(* IEC 61131-3 sources: PortalRobot/Portal_robot/Device/application/FB, 34 files *)

(* ---- FB_ALARM_MANAGER.st ---- *)
FUNCTION_BLOCK FB_ALARM_MANAGER
VAR_INPUT
	xResetAll      : BOOL; // Общий сброс ошибок ячейки
	xResetWarnings : BOOL; // Сброс накопленных предупреждений
END_VAR
VAR_IN_OUT
	Sources : ARRAY [1..13] OF ST_ALARM_SOURCE_DATA; // Унифицированные данные функциональных блоков
END_VAR
VAR_OUTPUT
	Status : ST_ALARM_STATUS; // Сводный статус журнала
	Events : ARRAY [1..100] OF ST_ALARM_EVENT; // Журнал активных и зафиксированных событий
END_VAR
VAR
	uiWriteIndex : UINT := 1; // Следующая ячейка кольцевого журнала
	udiSequence  : UDINT; // Общий порядковый номер события
	adwPreviousAlarm : ARRAY [1..13] OF DWORD; // Опубликованные аварии прошлого цикла
	audiPreviousWarning : ARRAY [1..13] OF UDINT; // Номера предупреждений прошлого цикла
	uiIndex : UINT; // Индекс источника или события
END_VAR

// --- BEGIN IMPLEMENTATION ---

// Предупреждения подтверждаются отдельно или вместе с общим сбросом.
IF xResetWarnings OR xResetAll THEN
	FOR uiIndex := 1 TO 100 DO
		IF Events[uiIndex].xActive
		AND (Events[uiIndex].eSeverity = E_ALARM_SEVERITY.WARNING) THEN
			Events[uiIndex].xActive := FALSE;
		END_IF;
	END_FOR;
END_IF;

// Менеджер не определяет причины: он регистрирует подготовленные данные владельцев блоков.
FOR uiIndex := 1 TO 13 DO
	UpdateSource(
		eSource := Sources[uiIndex].eSource,
		dwCurrent := Sources[uiIndex].dwAlarmActive,
		dwPrevious := adwPreviousAlarm[uiIndex]
	);

	IF Sources[uiIndex].stWarning.udiSequence <> audiPreviousWarning[uiIndex] THEN
		IF (Sources[uiIndex].stWarning.udiSequence <> UDINT#0)
		AND (Sources[uiIndex].stWarning.uiCode <> UINT#0) THEN
			AddEvent(
				eSource := Sources[uiIndex].eSource,
				eSeverity := E_ALARM_SEVERITY.WARNING,
				uiCode := Sources[uiIndex].stWarning.uiCode
			);
		END_IF;
		audiPreviousWarning[uiIndex] := Sources[uiIndex].stWarning.udiSequence;
	END_IF;
END_FOR;

Status.uiActiveAlarmCount := 0;
Status.uiActiveWarningCount := 0;
Status.uiHistoryCount := 0;

FOR uiIndex := 1 TO 100 DO
	IF Events[uiIndex].udiSequence <> UDINT#0 THEN
		Status.uiHistoryCount := Status.uiHistoryCount + 1;
	END_IF;
	IF Events[uiIndex].xActive THEN
		IF Events[uiIndex].eSeverity = E_ALARM_SEVERITY.ALARM THEN
			Status.uiActiveAlarmCount := Status.uiActiveAlarmCount + 1;
		ELSE
			Status.uiActiveWarningCount := Status.uiActiveWarningCount + 1;
		END_IF;
	END_IF;
END_FOR;

Status.uiActiveEventCount := Status.uiActiveAlarmCount + Status.uiActiveWarningCount;
Status.xAlarmActive := Status.uiActiveAlarmCount > 0;
Status.xWarningActive := Status.uiActiveWarningCount > 0;

(* ---- FB_AXIS.st ---- *)
FUNCTION_BLOCK FB_Axis
VAR_IN_OUT
    Axis     : AXIS_REF_SM3;   // ссылка на ось SoftMotion
    AxisData : ST_AXIS;        // все данные оси (команды, параметры, статусы)
END_VAR

VAR CONSTANT
    // ==================================================
    // Ошибки оси, MC-блоков и SoftMotion
    // ==================================================
    AXE_MC_POWER_ERROR       : DWORD := DWORD#16#00000001; // Ошибка MC_Power
    AXE_MC_RESET_ERROR       : DWORD := DWORD#16#00000002; // Ошибка MC_Reset
    AXE_MC_STOP_ERROR        : DWORD := DWORD#16#00000004; // Ошибка MC_Stop
    AXE_MC_JOG_ERROR         : DWORD := DWORD#16#00000008; // Ошибка MC_Jog
    AXE_MC_HOME_ERROR        : DWORD := DWORD#16#00000010; // Ошибка MC_Home
    AXE_MC_MOVE_ABS_ERROR    : DWORD := DWORD#16#00000020; // Ошибка абсолютного перемещения
    AXE_MC_MOVE_REL_ERROR    : DWORD := DWORD#16#00000040; // Ошибка относительного перемещения
    AXE_READ_POS_ERROR       : DWORD := DWORD#16#00000080; // Ошибка чтения позиции
    AXE_READ_STATUS_ERROR    : DWORD := DWORD#16#00000100; // Ошибка чтения статуса
    AXE_ERRORSTOP            : DWORD := DWORD#16#00000200; // Ось находится в ErrorStop
    AXE_FB_ERROR_OCCURRED    : DWORD := DWORD#16#00000400; // SoftMotion сообщил внутреннюю ошибку
    AXE_COMMAND_ABORTED      : DWORD := DWORD#16#00000800; // Команда движения прервана
    AXE_UNKNOWN_ACTUAL_ERROR : DWORD := DWORD#16#00001000; // Неизвестная текущая ошибка
    AXE_DRIVE_AXIS_ERROR     : DWORD := DWORD#16#00002000; // Ошибка привода

    // ==================================================
    // Логические ошибки блока
    // ==================================================
    LOG_POWER_PERMIT_LOST    : DWORD := DWORD#16#00000001; // Снято разрешение питания
    LOG_GLOBAL_DURING_POWER  : DWORD := DWORD#16#00000002; // Глобальная ошибка при включении
    LOG_GLOBAL_DURING_READY  : DWORD := DWORD#16#00000004; // Глобальная ошибка в готовности
    LOG_GLOBAL_DURING_MOTION : DWORD := DWORD#16#00000008; // Глобальная ошибка при движении
    LOG_JOG_CONFLICT         : DWORD := DWORD#16#00000010; // Одновременно заданы Jog+ и Jog-
    LOG_MOVE_ABS_NOT_HOMED   : DWORD := DWORD#16#00000020; // Абсолютное движение без поиска дома
    LOG_MOVE_REL_NOT_HOMED   : DWORD := DWORD#16#00000040; // Относительное движение без поиска дома
    LOG_STEP_TIMEOUT         : DWORD := DWORD#16#00000080; // Превышено время шага
    LOG_UNKNOWN_STEP         : DWORD := DWORD#16#00000100; // Неизвестный шаг автомата

    // ==================================================
    // Предупреждения блока
    // ==================================================
    WRN_NO_POWER_PERMIT : DWORD := DWORD#16#00000001; // Нет разрешения подачи питания

    MASK_LOCAL_LOGICAL_ERROR : DWORD :=
        LOG_JOG_CONFLICT OR
        LOG_MOVE_ABS_NOT_HOMED OR
        LOG_MOVE_REL_NOT_HOMED OR
        LOG_STEP_TIMEOUT OR
        LOG_UNKNOWN_STEP; // Логические первопричины, принадлежащие оси
END_VAR

VAR
    // Триггеры на команды
    rtEnable            : R_TRIG; // Фронт команды включения
    rtDisable           : R_TRIG; // Фронт команды отключения
    rtResetAllError     : R_TRIG; // Фронт общего сброса
    rtResetAxisError    : R_TRIG; // Фронт сброса привода
    rtResetLogicalError : R_TRIG; // Фронт сброса логики
    rtStop              : R_TRIG; // Фронт команды остановки
    rtHome              : R_TRIG; // Фронт команды поиска дома
    rtMoveAbsolute      : R_TRIG; // Фронт абсолютного перемещения
    rtMoveRelative      : R_TRIG; // Фронт относительного перемещения

    // Экземпляры MC-блоков
    fbPower        : MC_Power; // Управление питанием привода
    fbReset        : MC_Reset; // Сброс ошибки привода
    fbStop         : MC_Stop; // Контролируемая остановка
    fbJog          : MC_Jog; // Толчковое движение
    fbHome         : MC_Home; // Поиск домашней позиции
    fbMoveAbsolute : MC_MoveAbsolute; // Абсолютное перемещение
    fbMoveRelative : MC_MoveRelative; // Относительное перемещение
    fbReadPosition : MC_ReadActualPosition; // Чтение текущей позиции
    fbReadStatus   : MC_ReadStatus; // Чтение состояния оси
    fbReadAxisError: MC_ReadAxisError; // Чтение кода ошибки привода

    // Внутренние управляющие флаги
    xPowerRequest    : BOOL; // Защёлкнутый запрос питания
    xResetExecute    : BOOL; // Выполняется сброс привода
    xStopExecute     : BOOL; // Выполняется остановка
    xHomeExecute     : BOOL; // Выполняется поиск дома
    xMoveAbsExecute  : BOOL; // Выполняется абсолютное перемещение
    xMoveRelExecute  : BOOL; // Выполняется относительное перемещение
    xJogForwardExec  : BOOL; // Выполняется Jog в положительную сторону
    xJogBackwardExec : BOOL; // Выполняется Jog в отрицательную сторону

    // Для таймера шага
    iPrevStep        : E_AXIS_STATE := E_AXIS_STATE.DISABLED; // Предыдущий шаг автомата
    xStepChanged     : BOOL; // Шаг изменился в текущем цикле
    xStepTimerEnable : BOOL; // Разрешение таймера шага
    tonStep          : TON; // Таймер времени на шаге
    tonStepTimeout   : TON; // Таймер превышения времени шага

    // Для удержания предупреждений
    tpWarningHold : TP; // Удержание предупреждения для отображения
    xWarningPulse : BOOL; // Импульс нового предупреждения

    // Вспомогательные флаги для сброса
    xDoResetAxis    : BOOL; // Требуется сброс ошибок привода
    xDoResetLogical : BOOL; // Требуется сброс логических ошибок
    xNeedMcReset    : BOOL; // Требуется вызов MC_Reset

    // Актуальная ошибка оси (на основе MC-блоков)
    xAxisErrorActual : BOOL; // Текущая ошибка по выходам MC-блоков
END_VAR

// --- BEGIN IMPLEMENTATION ---

// ======================================================
// 1. ФРОНТЫ (триггеры на команды из структуры)
// ======================================================
rtEnable(CLK := AxisData.Command.xEnable);
rtDisable(CLK := AxisData.Command.xDisable);
rtResetAllError(CLK := AxisData.Command.xResetAllError);
rtResetAxisError(CLK := AxisData.Command.xResetAxisError);
rtResetLogicalError(CLK := AxisData.Command.xResetLogicalError);
rtStop(CLK := AxisData.Command.xStop);
rtHome(CLK := AxisData.Command.xHome);
rtMoveAbsolute(CLK := AxisData.Command.xMoveAbsolute);
rtMoveRelative(CLK := AxisData.Command.xMoveRelative);

// ======================================================
// 2. СТАТУСЫ ОТ MC-БЛОКОВ (запись в структуру)
// ======================================================
AxisData.Status.xPowered := fbPower.Status;

AxisData.Status.xLocalError :=
    fbPower.Error OR
    fbReset.Error OR
    fbStop.Error OR
    fbJog.Error OR
    fbHome.Error OR
    fbMoveAbsolute.Error OR
    fbMoveRelative.Error OR
    fbReadPosition.Error OR
    fbReadStatus.Error OR
    fbReadStatus.Errorstop OR
    fbReadStatus.FBErrorOccured;

AxisData.Status.xMotionBusy :=
    fbStop.Busy OR
    fbJog.Busy OR
    fbHome.Busy OR
    fbMoveAbsolute.Busy OR
    fbMoveRelative.Busy;

// MC_Reset нужен только для аппаратных/SoftMotion ошибок
xNeedMcReset := fbReadStatus.Errorstop OR fbReadStatus.FBErrorOccured OR fbReadAxisError.AxisError;

AxisData.Error.dwAxisError := AxisData.Error.dwAxisErrorActual OR AxisData.Error.dwAxisErrorLatched;
AxisData.Error.dwLogicalError := AxisData.Error.dwLogicalErrorLatched;
AxisData.Error.dwAllError := AxisData.Error.dwAxisError OR AxisData.Error.dwLogicalError;

// ======================================================
// 3. ЗНАЧЕНИЯ ПО УМОЛЧАНИЮ ДЛЯ ИСПОЛНИТЕЛЬНЫХ ФЛАГОВ
// ======================================================
xResetExecute    := FALSE;
xStopExecute     := FALSE;
xHomeExecute     := FALSE;
xMoveAbsExecute  := FALSE;
xMoveRelExecute  := FALSE;
xJogForwardExec  := FALSE;
xJogBackwardExec := FALSE;

AxisData.Status.xDone := FALSE;
xWarningPulse := FALSE;

// ======================================================
// 4. КОНЕЧНЫЙ АВТОМАТ (используем перечисление E_AXIS_STATE)
// ======================================================
CASE AxisData.Diag.iStep OF

    // --------------------------------------------------
    E_AXIS_STATE.DISABLED:
    // --------------------------------------------------
        AxisData.Diag.sStepName := 'DISABLED';
        AxisData.Diag.sWaitReason := 'Waiting Enable command';
        AxisData.Diag.tStepPreset := T#0S;

        xPowerRequest := FALSE;
        AxisData.Status.xHomed := FALSE;

        IF AxisData.Status.xError THEN
            AxisData.Diag.iStep := E_AXIS_STATE.ERROR_RESET_MANAGER;

        ELSIF rtEnable.Q AND NOT AxisData.Command.xPowerPermit THEN
            AxisData.Error.dwWarningLatched :=
                AxisData.Error.dwWarningLatched OR WRN_NO_POWER_PERMIT;
            AxisData.Diag.sWarningText := 'Нет разрешения на запуск двигателя';
            AxisData.Diag.stWarning.uiCode := UINT#1;
            AxisData.Diag.stWarning.udiSequence := AxisData.Diag.stWarning.udiSequence + UDINT#1;
            IF AxisData.Diag.stWarning.udiSequence = UDINT#0 THEN
                AxisData.Diag.stWarning.udiSequence := UDINT#1;
            END_IF;
            xWarningPulse := TRUE;
            AxisData.Diag.sWaitReason := 'Power permit missing';

        ELSIF NOT AxisData.Command.xPowerPermit THEN
            AxisData.Diag.sWaitReason := 'Power permit missing';

        ELSIF rtEnable.Q THEN
            xPowerRequest := TRUE;
            AxisData.Diag.iStep := E_AXIS_STATE.POWERING;
        END_IF;

    // --------------------------------------------------
    E_AXIS_STATE.POWERING:
    // --------------------------------------------------
        AxisData.Diag.sStepName := 'POWERING';
        AxisData.Diag.sWaitReason := 'Waiting MC_Power.Status';
        AxisData.Diag.tStepPreset := AxisData.Timeouts.tPowerTimeout;

        xPowerRequest := TRUE;

        IF NOT AxisData.Command.xPowerPermit THEN
            xPowerRequest := FALSE;
            AxisData.Error.dwLogicalErrorLatched :=
                AxisData.Error.dwLogicalErrorLatched OR LOG_POWER_PERMIT_LOST;
            AxisData.Diag.iLastErrorStep := TO_INT(AxisData.Diag.iStep);
            AxisData.Diag.iStep := E_AXIS_STATE.ERROR_RESET_MANAGER;

        ELSIF AxisData.Command.xGlobalError THEN
            xPowerRequest := FALSE;
            AxisData.Error.dwLogicalErrorLatched :=
                AxisData.Error.dwLogicalErrorLatched OR LOG_GLOBAL_DURING_POWER;
            AxisData.Diag.iLastErrorStep := TO_INT(AxisData.Diag.iStep);
            AxisData.Diag.iStep := E_AXIS_STATE.ERROR_RESET_MANAGER;

        ELSIF fbPower.Error THEN
            xPowerRequest := FALSE;
            AxisData.Error.dwAxisErrorLatched :=
                AxisData.Error.dwAxisErrorLatched OR AXE_MC_POWER_ERROR;
            AxisData.Diag.udiLastErrorID := TO_UDINT(fbPower.ErrorID);
            AxisData.Diag.iLastErrorStep := TO_INT(AxisData.Diag.iStep);
            AxisData.Diag.iStep := E_AXIS_STATE.ERROR_RESET_MANAGER;

        ELSIF fbPower.Status THEN
            AxisData.Diag.iStep := E_AXIS_STATE.READY;

        ELSIF rtDisable.Q THEN
            xPowerRequest := FALSE;
            AxisData.Diag.iStep := E_AXIS_STATE.DISABLED;
        END_IF;

    // --------------------------------------------------
    E_AXIS_STATE.READY:
    // --------------------------------------------------
        AxisData.Diag.sStepName := 'READY';
        AxisData.Diag.sWaitReason := 'Waiting command';
        AxisData.Diag.tStepPreset := T#0S;

        xPowerRequest := TRUE;

        IF NOT AxisData.Command.xPowerPermit THEN
            xPowerRequest := FALSE;
            AxisData.Diag.iStep := E_AXIS_STATE.DISABLED;

        ELSIF rtDisable.Q THEN
            xPowerRequest := FALSE;
            AxisData.Diag.iStep := E_AXIS_STATE.DISABLED;

        ELSIF AxisData.Command.xGlobalError THEN
            AxisData.Error.dwLogicalErrorLatched :=
                AxisData.Error.dwLogicalErrorLatched OR LOG_GLOBAL_DURING_READY;
            AxisData.Diag.iLastErrorStep := TO_INT(AxisData.Diag.iStep);
            AxisData.Diag.iStep := E_AXIS_STATE.ERROR_RESET_MANAGER;

        ELSIF xAxisErrorActual THEN
            AxisData.Error.dwAxisErrorLatched :=
                AxisData.Error.dwAxisErrorLatched OR AxisData.Error.dwAxisErrorActual;
            AxisData.Diag.iLastErrorStep := TO_INT(AxisData.Diag.iStep);
            AxisData.Diag.iStep := E_AXIS_STATE.ERROR_RESET_MANAGER;

        ELSIF AxisData.Command.xJogPositive AND AxisData.Command.xJogNegative THEN
            AxisData.Error.dwLogicalErrorLatched :=
                AxisData.Error.dwLogicalErrorLatched OR LOG_JOG_CONFLICT;
            AxisData.Diag.iLastErrorStep := TO_INT(AxisData.Diag.iStep);
            AxisData.Diag.iStep := E_AXIS_STATE.ERROR_RESET_MANAGER;

        ELSIF AxisData.Command.xJogPositive OR AxisData.Command.xJogNegative THEN
            AxisData.Diag.iStep := E_AXIS_STATE.JOGGING;

        ELSIF rtHome.Q THEN
            AxisData.Diag.iStep := E_AXIS_STATE.HOMING;

        ELSIF rtMoveAbsolute.Q THEN
            IF AxisData.Status.xHomed THEN
                AxisData.Diag.iStep := E_AXIS_STATE.MOVE_ABSOLUTE;
            ELSE
                AxisData.Error.dwLogicalErrorLatched :=
                    AxisData.Error.dwLogicalErrorLatched OR LOG_MOVE_ABS_NOT_HOMED;
                AxisData.Diag.iLastErrorStep := TO_INT(AxisData.Diag.iStep);
                AxisData.Diag.iStep := E_AXIS_STATE.ERROR_RESET_MANAGER;
            END_IF;

        ELSIF rtMoveRelative.Q THEN
            IF AxisData.Status.xHomed THEN
                AxisData.Diag.iStep := E_AXIS_STATE.MOVE_RELATIVE;
            ELSE
                AxisData.Error.dwLogicalErrorLatched :=
                    AxisData.Error.dwLogicalErrorLatched OR LOG_MOVE_REL_NOT_HOMED;
                AxisData.Diag.iLastErrorStep := TO_INT(AxisData.Diag.iStep);
                AxisData.Diag.iStep := E_AXIS_STATE.ERROR_RESET_MANAGER;
            END_IF;
        END_IF;

    // --------------------------------------------------
    E_AXIS_STATE.JOGGING:
    // --------------------------------------------------
        AxisData.Diag.sStepName := 'JOGGING';
        AxisData.Diag.sWaitReason := 'Jog active';
        AxisData.Diag.tStepPreset := T#0S;

        xPowerRequest := TRUE;
        xJogForwardExec  := AxisData.Command.xJogPositive AND NOT AxisData.Command.xJogNegative;
        xJogBackwardExec := AxisData.Command.xJogNegative AND NOT AxisData.Command.xJogPositive;

        IF NOT AxisData.Command.xPowerPermit THEN
            xJogForwardExec := FALSE;
            xJogBackwardExec := FALSE;
            AxisData.Error.dwLogicalErrorLatched :=
                AxisData.Error.dwLogicalErrorLatched OR LOG_POWER_PERMIT_LOST;
            AxisData.Diag.iLastErrorStep := TO_INT(AxisData.Diag.iStep);
            AxisData.Diag.iStep := E_AXIS_STATE.STOPPING;

        ELSIF AxisData.Command.xGlobalError THEN
            xJogForwardExec := FALSE;
            xJogBackwardExec := FALSE;
            AxisData.Error.dwLogicalErrorLatched :=
                AxisData.Error.dwLogicalErrorLatched OR LOG_GLOBAL_DURING_MOTION;
            AxisData.Diag.iLastErrorStep := TO_INT(AxisData.Diag.iStep);
            AxisData.Diag.iStep := E_AXIS_STATE.STOPPING;

        ELSIF xAxisErrorActual THEN
            xJogForwardExec := FALSE;
            xJogBackwardExec := FALSE;
            AxisData.Error.dwAxisErrorLatched :=
                AxisData.Error.dwAxisErrorLatched OR AxisData.Error.dwAxisErrorActual;
            AxisData.Diag.iLastErrorStep := TO_INT(AxisData.Diag.iStep);
            AxisData.Diag.iStep := E_AXIS_STATE.STOPPING;

        ELSIF rtStop.Q THEN
            xJogForwardExec := FALSE;
            xJogBackwardExec := FALSE;
            AxisData.Diag.iStep := E_AXIS_STATE.STOPPING;

        ELSIF AxisData.Command.xJogPositive AND AxisData.Command.xJogNegative THEN
            xJogForwardExec := FALSE;
            xJogBackwardExec := FALSE;
            AxisData.Error.dwLogicalErrorLatched :=
                AxisData.Error.dwLogicalErrorLatched OR LOG_JOG_CONFLICT;
            AxisData.Diag.iLastErrorStep := TO_INT(AxisData.Diag.iStep);
            AxisData.Diag.iStep := E_AXIS_STATE.STOPPING;

        ELSIF NOT AxisData.Command.xJogPositive AND NOT AxisData.Command.xJogNegative THEN
            xJogForwardExec := FALSE;
            xJogBackwardExec := FALSE;
            AxisData.Diag.iStep := E_AXIS_STATE.READY;
        END_IF;

    // --------------------------------------------------
    E_AXIS_STATE.HOMING:
    // --------------------------------------------------
        AxisData.Diag.sStepName := 'HOMING';
        AxisData.Diag.sWaitReason := 'Waiting MC_Home.Done';
        AxisData.Diag.tStepPreset := AxisData.Timeouts.tHomeTimeout;

        xPowerRequest := TRUE;
        xHomeExecute := TRUE;

        IF NOT AxisData.Command.xPowerPermit THEN
            xHomeExecute := FALSE;
            AxisData.Error.dwLogicalErrorLatched :=
                AxisData.Error.dwLogicalErrorLatched OR LOG_POWER_PERMIT_LOST;
            AxisData.Diag.iLastErrorStep := TO_INT(AxisData.Diag.iStep);
            AxisData.Diag.iStep := E_AXIS_STATE.STOPPING;

        ELSIF AxisData.Command.xGlobalError THEN
            xHomeExecute := FALSE;
            AxisData.Error.dwLogicalErrorLatched :=
                AxisData.Error.dwLogicalErrorLatched OR LOG_GLOBAL_DURING_MOTION;
            AxisData.Diag.iLastErrorStep := TO_INT(AxisData.Diag.iStep);
            AxisData.Diag.iStep := E_AXIS_STATE.STOPPING;

        ELSIF rtStop.Q THEN
            xHomeExecute := FALSE;
            AxisData.Diag.iStep := E_AXIS_STATE.STOPPING;

        ELSIF fbHome.Error THEN
            xHomeExecute := FALSE;
            AxisData.Error.dwAxisErrorLatched :=
                AxisData.Error.dwAxisErrorLatched OR AXE_MC_HOME_ERROR;
            AxisData.Diag.udiLastErrorID := TO_UDINT(fbHome.ErrorID);
            AxisData.Diag.iLastErrorStep := TO_INT(AxisData.Diag.iStep);
            AxisData.Diag.iStep := E_AXIS_STATE.ERROR_RESET_MANAGER;

        ELSIF fbHome.CommandAborted THEN
            xHomeExecute := FALSE;
            AxisData.Error.dwAxisErrorLatched :=
                AxisData.Error.dwAxisErrorLatched OR AXE_COMMAND_ABORTED;
            AxisData.Diag.udiLastErrorID := 3003;
            AxisData.Diag.iLastErrorStep := TO_INT(AxisData.Diag.iStep);
            AxisData.Diag.iStep := E_AXIS_STATE.ERROR_RESET_MANAGER;

        ELSIF xAxisErrorActual THEN
            xHomeExecute := FALSE;
            AxisData.Error.dwAxisErrorLatched :=
                AxisData.Error.dwAxisErrorLatched OR AxisData.Error.dwAxisErrorActual;
            AxisData.Diag.iLastErrorStep := TO_INT(AxisData.Diag.iStep);
            AxisData.Diag.iStep := E_AXIS_STATE.ERROR_RESET_MANAGER;

        ELSIF fbHome.Done THEN
            xHomeExecute := FALSE;
            AxisData.Status.xHomed := TRUE;
            AxisData.Status.xDone := TRUE;
            AxisData.Diag.iStep := E_AXIS_STATE.READY;
        END_IF;

    // --------------------------------------------------
    E_AXIS_STATE.MOVE_ABSOLUTE:
    // --------------------------------------------------
        AxisData.Diag.sStepName := 'MOVING_ABSOLUTE';
        AxisData.Diag.sWaitReason := 'Waiting MC_MoveAbsolute.Done';
        AxisData.Diag.tStepPreset := AxisData.Timeouts.tMoveTimeout;

        xPowerRequest := TRUE;
        xMoveAbsExecute := TRUE;

        IF NOT AxisData.Command.xPowerPermit THEN
            xMoveAbsExecute := FALSE;
            AxisData.Error.dwLogicalErrorLatched :=
                AxisData.Error.dwLogicalErrorLatched OR LOG_POWER_PERMIT_LOST;
            AxisData.Diag.iLastErrorStep := TO_INT(AxisData.Diag.iStep);
            AxisData.Diag.iStep := E_AXIS_STATE.STOPPING;

        ELSIF AxisData.Command.xGlobalError THEN
            xMoveAbsExecute := FALSE;
            AxisData.Error.dwLogicalErrorLatched :=
                AxisData.Error.dwLogicalErrorLatched OR LOG_GLOBAL_DURING_MOTION;
            AxisData.Diag.iLastErrorStep := TO_INT(AxisData.Diag.iStep);
            AxisData.Diag.iStep := E_AXIS_STATE.STOPPING;

        ELSIF rtStop.Q THEN
            xMoveAbsExecute := FALSE;
            AxisData.Diag.iStep := E_AXIS_STATE.STOPPING;

        ELSIF fbMoveAbsolute.Error THEN
            xMoveAbsExecute := FALSE;
            AxisData.Error.dwAxisErrorLatched :=
                AxisData.Error.dwAxisErrorLatched OR AXE_MC_MOVE_ABS_ERROR;
            AxisData.Diag.udiLastErrorID := TO_UDINT(fbMoveAbsolute.ErrorID);
            AxisData.Diag.iLastErrorStep := TO_INT(AxisData.Diag.iStep);
            AxisData.Diag.iStep := E_AXIS_STATE.ERROR_RESET_MANAGER;

        ELSIF fbMoveAbsolute.CommandAborted THEN
            xMoveAbsExecute := FALSE;
            AxisData.Error.dwAxisErrorLatched :=
                AxisData.Error.dwAxisErrorLatched OR AXE_COMMAND_ABORTED;
            AxisData.Diag.udiLastErrorID := 3003;
            AxisData.Diag.iLastErrorStep := TO_INT(AxisData.Diag.iStep);
            AxisData.Diag.iStep := E_AXIS_STATE.ERROR_RESET_MANAGER;

        ELSIF xAxisErrorActual THEN
            xMoveAbsExecute := FALSE;
            AxisData.Error.dwAxisErrorLatched :=
                AxisData.Error.dwAxisErrorLatched OR AxisData.Error.dwAxisErrorActual;
            AxisData.Diag.iLastErrorStep := TO_INT(AxisData.Diag.iStep);
            AxisData.Diag.iStep := E_AXIS_STATE.ERROR_RESET_MANAGER;

        ELSIF fbMoveAbsolute.Done THEN
            xMoveAbsExecute := FALSE;
            AxisData.Status.xDone := TRUE;
            AxisData.Diag.iStep := E_AXIS_STATE.READY;
        END_IF;

    // --------------------------------------------------
    E_AXIS_STATE.MOVE_RELATIVE:
    // --------------------------------------------------
        AxisData.Diag.sStepName := 'MOVING_RELATIVE';
        AxisData.Diag.sWaitReason := 'Waiting MC_MoveRelative.Done';
        AxisData.Diag.tStepPreset := AxisData.Timeouts.tMoveTimeout;

        xPowerRequest := TRUE;
        xMoveRelExecute := TRUE;

        IF NOT AxisData.Command.xPowerPermit THEN
            xMoveRelExecute := FALSE;
            AxisData.Error.dwLogicalErrorLatched :=
                AxisData.Error.dwLogicalErrorLatched OR LOG_POWER_PERMIT_LOST;
            AxisData.Diag.iLastErrorStep := TO_INT(AxisData.Diag.iStep);
            AxisData.Diag.iStep := E_AXIS_STATE.STOPPING;

        ELSIF AxisData.Command.xGlobalError THEN
            xMoveRelExecute := FALSE;
            AxisData.Error.dwLogicalErrorLatched :=
                AxisData.Error.dwLogicalErrorLatched OR LOG_GLOBAL_DURING_MOTION;
            AxisData.Diag.iLastErrorStep := TO_INT(AxisData.Diag.iStep);
            AxisData.Diag.iStep := E_AXIS_STATE.STOPPING;

        ELSIF rtStop.Q THEN
            xMoveRelExecute := FALSE;
            AxisData.Diag.iStep := E_AXIS_STATE.STOPPING;

        ELSIF fbMoveRelative.Error THEN
            xMoveRelExecute := FALSE;
            AxisData.Error.dwAxisErrorLatched :=
                AxisData.Error.dwAxisErrorLatched OR AXE_MC_MOVE_REL_ERROR;
            AxisData.Diag.udiLastErrorID := TO_UDINT(fbMoveRelative.ErrorID);
            AxisData.Diag.iLastErrorStep := TO_INT(AxisData.Diag.iStep);
            AxisData.Diag.iStep := E_AXIS_STATE.ERROR_RESET_MANAGER;

        ELSIF fbMoveRelative.CommandAborted THEN
            xMoveRelExecute := FALSE;
            AxisData.Error.dwAxisErrorLatched :=
                AxisData.Error.dwAxisErrorLatched OR AXE_COMMAND_ABORTED;
            AxisData.Diag.udiLastErrorID := 3003;
            AxisData.Diag.iLastErrorStep := TO_INT(AxisData.Diag.iStep);
            AxisData.Diag.iStep := E_AXIS_STATE.ERROR_RESET_MANAGER;

        ELSIF xAxisErrorActual THEN
            xMoveRelExecute := FALSE;
            AxisData.Error.dwAxisErrorLatched :=
                AxisData.Error.dwAxisErrorLatched OR AxisData.Error.dwAxisErrorActual;
            AxisData.Diag.iLastErrorStep := TO_INT(AxisData.Diag.iStep);
            AxisData.Diag.iStep := E_AXIS_STATE.ERROR_RESET_MANAGER;

        ELSIF fbMoveRelative.Done THEN
            xMoveRelExecute := FALSE;
            AxisData.Status.xDone := TRUE;
            AxisData.Diag.iStep := E_AXIS_STATE.READY;
        END_IF;

    // --------------------------------------------------
    E_AXIS_STATE.STOPPING:
    // --------------------------------------------------
        AxisData.Diag.sStepName := 'STOPPING';
        AxisData.Diag.sWaitReason := 'Waiting MC_Stop.Done';
        AxisData.Diag.tStepPreset := AxisData.Timeouts.tStopTimeout;

        xPowerRequest := TRUE;
        xStopExecute := TRUE;

        IF fbStop.Error THEN
            xStopExecute := FALSE;
            AxisData.Error.dwAxisErrorLatched :=
                AxisData.Error.dwAxisErrorLatched OR AXE_MC_STOP_ERROR;
            AxisData.Diag.udiLastErrorID := TO_UDINT(fbStop.ErrorID);
            AxisData.Diag.iLastErrorStep := TO_INT(AxisData.Diag.iStep);
            AxisData.Diag.iStep := E_AXIS_STATE.ERROR_RESET_MANAGER;

        ELSIF fbStop.Done THEN
            AxisData.Status.xDone := TRUE;
            AxisData.Diag.iStep := E_AXIS_STATE.STOP_RELEASE;
        END_IF;

    // --------------------------------------------------
    E_AXIS_STATE.STOP_RELEASE:
    // --------------------------------------------------
        AxisData.Diag.sStepName := 'STOP_RELEASE';
        AxisData.Diag.sWaitReason := 'Releasing MC_Stop.Execute';
        AxisData.Diag.tStepPreset := T#1S;

        xPowerRequest := TRUE;
        xStopExecute := FALSE;

        IF NOT fbStop.Busy THEN
            IF AxisData.Command.xGlobalError OR
               (AxisData.Error.dwAxisErrorLatched <> DWORD#0) OR
               (AxisData.Error.dwLogicalErrorLatched <> DWORD#0) OR
               xAxisErrorActual
            THEN
                AxisData.Diag.iStep := E_AXIS_STATE.ERROR_RESET_MANAGER;
            ELSE
                AxisData.Diag.iStep := E_AXIS_STATE.READY;
            END_IF;
        END_IF;

    // --------------------------------------------------
    E_AXIS_STATE.ERROR_RESET_MANAGER:
    // --------------------------------------------------
        AxisData.Diag.sStepName := 'ERROR';
        AxisData.Diag.tStepPreset := T#0S;

        xResetExecute    := FALSE;
        xStopExecute     := FALSE;
        xHomeExecute     := FALSE;
        xMoveAbsExecute  := FALSE;
        xMoveRelExecute  := FALSE;
        xJogForwardExec  := FALSE;
        xJogBackwardExec := FALSE;

        IF AxisData.Timeouts.xDisableOnError THEN
            xPowerRequest := FALSE;
        ELSE
            xPowerRequest := AxisData.Command.xPowerPermit AND NOT xAxisErrorActual;
        END_IF;

        IF (AxisData.Error.dwAxisError = DWORD#0) AND
           (AxisData.Error.dwLogicalError = DWORD#0) AND
           NOT AxisData.Command.xGlobalError
        THEN
            AxisData.Diag.iStep := E_AXIS_STATE.DISABLED;

        ELSE
            IF AxisData.Command.xGlobalError THEN
                AxisData.Diag.sWaitReason := 'Waiting global error release';
            ELSIF (AxisData.Error.dwAxisError <> DWORD#0) AND
                  (AxisData.Error.dwLogicalError <> DWORD#0) THEN
                AxisData.Diag.sWaitReason := 'Waiting ResetAllError';
            ELSIF AxisData.Error.dwAxisError <> DWORD#0 THEN
                AxisData.Diag.sWaitReason := 'Waiting ResetAxisError or ResetAllError';
            ELSIF AxisData.Error.dwLogicalError <> DWORD#0 THEN
                AxisData.Diag.sWaitReason := 'Waiting ResetLogicalError or ResetAllError';
            ELSE
                AxisData.Diag.sWaitReason := 'Waiting reset';
            END_IF;

            IF rtResetAllError.Q THEN
                xDoResetAxis := TRUE;
                xDoResetLogical := TRUE;
                IF xNeedMcReset THEN
                    AxisData.Diag.iStep := E_AXIS_STATE.RESET_AXIS_ERROR;
                ELSE
                    AxisData.Diag.iStep := E_AXIS_STATE.RESET_FINISH;
                END_IF;

            ELSIF rtResetAxisError.Q THEN
                xDoResetAxis := TRUE;
                xDoResetLogical := FALSE;
                IF xNeedMcReset THEN
                    AxisData.Diag.iStep := E_AXIS_STATE.RESET_AXIS_ERROR;
                ELSE
                    AxisData.Diag.iStep := E_AXIS_STATE.RESET_FINISH;
                END_IF;

            ELSIF rtResetLogicalError.Q THEN
                xDoResetAxis := FALSE;
                xDoResetLogical := TRUE;
                AxisData.Diag.iStep := E_AXIS_STATE.RESET_FINISH;
            END_IF;
        END_IF;

    // --------------------------------------------------
    E_AXIS_STATE.RESET_AXIS_ERROR:
    // --------------------------------------------------
        AxisData.Diag.sStepName := 'RESET_AXIS_ERROR';
        AxisData.Diag.sWaitReason := 'Waiting MC_Reset.Done';
        AxisData.Diag.tStepPreset := AxisData.Timeouts.tResetTimeout;

        xPowerRequest := FALSE;
        xResetExecute := TRUE;

        IF fbReset.Error THEN
            xResetExecute := FALSE;
            AxisData.Error.dwAxisErrorLatched :=
                AxisData.Error.dwAxisErrorLatched OR AXE_MC_RESET_ERROR;
            AxisData.Diag.udiLastErrorID := TO_UDINT(fbReset.ErrorID);
            AxisData.Diag.iLastErrorStep := TO_INT(AxisData.Diag.iStep);
            AxisData.Diag.iStep := E_AXIS_STATE.ERROR_RESET_MANAGER;

        ELSIF fbReset.Done THEN
            xResetExecute := FALSE;
            AxisData.Diag.iStep := E_AXIS_STATE.RESET_RELEASE;
        END_IF;

    // --------------------------------------------------
    E_AXIS_STATE.RESET_RELEASE:
    // --------------------------------------------------
        AxisData.Diag.sStepName := 'RESET_RELEASE';
        AxisData.Diag.sWaitReason := 'Releasing MC_Reset.Execute';
        AxisData.Diag.tStepPreset := T#1S;

        xPowerRequest := FALSE;
        xResetExecute := FALSE;

        IF NOT fbReset.Busy THEN
            AxisData.Diag.iStep := E_AXIS_STATE.RESET_FINISH;
        END_IF;

    // --------------------------------------------------
    E_AXIS_STATE.RESET_FINISH:
    // --------------------------------------------------
        AxisData.Diag.sStepName := 'RESET_FINISH';
        AxisData.Diag.sWaitReason := 'Finishing reset';
        AxisData.Diag.tStepPreset := T#0S;

        xPowerRequest := FALSE;
        xResetExecute := FALSE;

        IF xDoResetAxis THEN
            AxisData.Error.dwAxisErrorLatched := DWORD#0;
        END_IF;
        IF xDoResetLogical THEN
            AxisData.Error.dwLogicalErrorLatched := DWORD#0;
            AxisData.Diag.xStepTimeout := FALSE;
        END_IF;

        xDoResetAxis := FALSE;
        xDoResetLogical := FALSE;

        // Финальная проверка
        IF AxisData.Error.dwAxisErrorActual <> DWORD#0 THEN
            AxisData.Error.dwAxisErrorLatched :=
                AxisData.Error.dwAxisErrorLatched OR AxisData.Error.dwAxisErrorActual;
            AxisData.Diag.iStep := E_AXIS_STATE.ERROR_RESET_MANAGER;

        ELSIF AxisData.Error.dwAxisErrorLatched <> DWORD#0 THEN
            AxisData.Diag.iStep := E_AXIS_STATE.ERROR_RESET_MANAGER;

        ELSIF AxisData.Error.dwLogicalErrorLatched <> DWORD#0 THEN
            AxisData.Diag.iStep := E_AXIS_STATE.ERROR_RESET_MANAGER;

        ELSIF AxisData.Command.xGlobalError THEN
            AxisData.Diag.iStep := E_AXIS_STATE.ERROR_RESET_MANAGER;

        ELSE
            AxisData.Diag.iStep := E_AXIS_STATE.DISABLED;
        END_IF;

    // --------------------------------------------------
    ELSE  // неизвестное состояние
    // --------------------------------------------------
        AxisData.Error.dwLogicalErrorLatched :=
            AxisData.Error.dwLogicalErrorLatched OR LOG_UNKNOWN_STEP;
        AxisData.Diag.iLastErrorStep := TO_INT(AxisData.Diag.iStep);
        AxisData.Diag.iStep := E_AXIS_STATE.ERROR_RESET_MANAGER;

END_CASE;

// ======================================================
// 5. ТАЙМЕР ШАГА И КОНТРОЛЬ ТАЙМАУТА
// ======================================================
xStepChanged := (AxisData.Diag.iStep <> iPrevStep);
IF xStepChanged THEN
    iPrevStep := AxisData.Diag.iStep;
    xStepTimerEnable := FALSE;
ELSE
    xStepTimerEnable := TRUE;
END_IF;

tonStep(IN := xStepTimerEnable, PT := T#1000H);
AxisData.Diag.tStepElapsed := tonStep.ET;

tonStepTimeout(
    IN := xStepTimerEnable AND (AxisData.Diag.tStepPreset > T#0S),
    PT := AxisData.Diag.tStepPreset
);

IF tonStepTimeout.Q AND (AxisData.Diag.iStep <> E_AXIS_STATE.ERROR_RESET_MANAGER) THEN
    AxisData.Diag.xStepTimeout := TRUE;
    AxisData.Error.dwLogicalErrorLatched := AxisData.Error.dwLogicalErrorLatched OR LOG_STEP_TIMEOUT;
    AxisData.Diag.iLastErrorStep := TO_INT(AxisData.Diag.iStep);

    xResetExecute    := FALSE;
    xStopExecute     := FALSE;
    xHomeExecute     := FALSE;
    xMoveAbsExecute  := FALSE;
    xMoveRelExecute  := FALSE;
    xJogForwardExec  := FALSE;
    xJogBackwardExec := FALSE;

    AxisData.Diag.iStep := E_AXIS_STATE.ERROR_RESET_MANAGER;
END_IF;

// ======================================================
// 6. УДЕРЖАНИЕ ПРЕДУПРЕЖДЕНИЙ (TP)
// ======================================================
tpWarningHold(IN := xWarningPulse, PT := T#2S);
IF NOT tpWarningHold.Q THEN
    AxisData.Error.dwWarningLatched := DWORD#0;
    AxisData.Diag.sWarningText := '';
END_IF;
AxisData.Error.dwWarning := AxisData.Error.dwWarningLatched;
AxisData.Status.xWarning := (AxisData.Error.dwWarning <> DWORD#0);

// ======================================================
// 7. ВЫЗОВ MC-БЛОКОВ
// ======================================================
fbPower(
    Axis := Axis,
    Enable := xPowerRequest,
    bRegulatorOn := xPowerRequest,
    bDriveStart := xPowerRequest
);

fbReset(
    Axis := Axis,
    Execute := xResetExecute
);

fbStop(
    Axis := Axis,
    Execute := xStopExecute,
    Deceleration := AxisData.MotionParam.lrDeceleration,
    Jerk := AxisData.MotionParam.lrJerk
);

fbJog(
    Axis := Axis,
    JogForward := xJogForwardExec,
    JogBackward := xJogBackwardExec,
    Velocity := AxisData.MotionParam.lrVelocity,
    Acceleration := AxisData.MotionParam.lrAcceleration,
    Deceleration := AxisData.MotionParam.lrDeceleration,
    Jerk := AxisData.MotionParam.lrJerk
);

fbHome(
    Axis := Axis,
    Execute := xHomeExecute,
    Position := AxisData.MotionParam.lrHomePosition
);

fbMoveAbsolute(
    Axis := Axis,
    Execute := xMoveAbsExecute,
    Position := AxisData.MotionParam.lrTargetPosition,
    Velocity := AxisData.MotionParam.lrVelocity,
    Acceleration := AxisData.MotionParam.lrAcceleration,
    Deceleration := AxisData.MotionParam.lrDeceleration,
    Jerk := AxisData.MotionParam.lrJerk,
    Direction := MC_DIRECTION.shortest,
    BufferMode := MC_BUFFER_MODE.Aborting
);

fbMoveRelative(
    Axis := Axis,
    Execute := xMoveRelExecute,
    Distance := AxisData.MotionParam.lrDistance,
    Velocity := AxisData.MotionParam.lrVelocity,
    Acceleration := AxisData.MotionParam.lrAcceleration,
    Deceleration := AxisData.MotionParam.lrDeceleration,
    Jerk := AxisData.MotionParam.lrJerk,
    BufferMode := MC_BUFFER_MODE.Aborting
);

fbReadPosition(
    Axis := Axis,
    Enable := TRUE
);

fbReadStatus(
    Axis := Axis,
    Enable := TRUE
);

fbReadAxisError(
    Axis := Axis,
    Enable := TRUE
);

// ======================================================
// 8. ИТОГОВЫЕ СТАТУСЫ (запись в структуру)
// ======================================================
AxisData.Status.lrActualPosition := LREAL_TO_REAL(fbReadPosition.Position);

// Повторно собираем актуальные ошибки (для полноты)
AxisData.Error.dwAxisErrorActual := DWORD#0;
AxisData.Error.dwAxisErrorActual.0  := fbPower.Error;
AxisData.Error.dwAxisErrorActual.1  := fbReset.Error;
AxisData.Error.dwAxisErrorActual.2  := fbStop.Error;
AxisData.Error.dwAxisErrorActual.3  := fbJog.Error;
AxisData.Error.dwAxisErrorActual.4  := fbHome.Error;
AxisData.Error.dwAxisErrorActual.5  := fbMoveAbsolute.Error;
AxisData.Error.dwAxisErrorActual.6  := fbMoveRelative.Error;
AxisData.Error.dwAxisErrorActual.7  := fbReadPosition.Error;
AxisData.Error.dwAxisErrorActual.8  := fbReadStatus.Error;
AxisData.Error.dwAxisErrorActual.9  := fbReadStatus.Errorstop;
AxisData.Error.dwAxisErrorActual.10 := fbReadStatus.FBErrorOccured;
AxisData.Error.dwAxisErrorActual.11 := fbReadAxisError.AxisError;

xAxisErrorActual := (AxisData.Error.dwAxisErrorActual <> DWORD#0);

AxisData.Status.xLocalError :=
    fbPower.Error OR
    fbReset.Error OR
    fbStop.Error OR
    fbJog.Error OR
    fbHome.Error OR
    fbMoveAbsolute.Error OR
    fbMoveRelative.Error OR
    fbReadPosition.Error OR
    fbReadStatus.Error OR
    fbReadStatus.Errorstop OR
    fbReadStatus.FBErrorOccured OR
    fbReadAxisError.AxisError;

AxisData.Status.xMotionBusy :=
    fbStop.Busy OR
    fbJog.Busy OR
    fbHome.Busy OR
    fbMoveAbsolute.Busy OR
    fbMoveRelative.Busy;

xNeedMcReset :=
    fbReadStatus.Errorstop OR
    fbReadStatus.FBErrorOccured OR
    fbReadAxisError.AxisError;

AxisData.Error.dwAxisError := AxisData.Error.dwAxisErrorActual OR AxisData.Error.dwAxisErrorLatched;
AxisData.Error.dwLogicalError := AxisData.Error.dwLogicalErrorLatched;
AxisData.Error.dwAllError := AxisData.Error.dwAxisError OR AxisData.Error.dwLogicalError;
AxisData.Error.dwAlarmActive := AxisData.Error.dwAxisError
    OR SHL(AxisData.Error.dwLogicalError AND MASK_LOCAL_LOGICAL_ERROR, 16);
AxisData.Error.dwDriveAxisErrorID := fbReadAxisError.AxisErrorID;

AxisData.Status.xAxisError := (AxisData.Error.dwAxisError <> DWORD#0);
AxisData.Status.xLogicalError := (AxisData.Error.dwLogicalError <> DWORD#0);
AxisData.Status.xAxisResetNeeded := AxisData.Status.xAxisError;
AxisData.Status.xLogicalResetNeeded := AxisData.Status.xLogicalError;

AxisData.Status.xError :=
    (AxisData.Diag.iStep = E_AXIS_STATE.ERROR_RESET_MANAGER) OR
    AxisData.Status.xAxisError OR
    AxisData.Status.xLogicalError OR
    AxisData.Command.xGlobalError;

AxisData.Status.xBusy :=
    fbPower.Busy OR
    fbReset.Busy OR
    AxisData.Status.xMotionBusy;

AxisData.Status.xCanStartMotion :=
    (AxisData.Diag.iStep = E_AXIS_STATE.READY) AND
    AxisData.Status.xPowered AND
    NOT AxisData.Status.xAxisError AND
    NOT AxisData.Status.xLogicalError AND
    NOT AxisData.Command.xGlobalError;

// ======================================================
// 9. ТЕКСТ ОШИБКИ И ID
// ======================================================
AxisData.Diag.sErrorText := '';
AxisData.Diag.udiActualErrorID := 0;

IF (AxisData.Error.dwLogicalError AND LOG_POWER_PERMIT_LOST) <> DWORD#0 THEN
    AxisData.Diag.sErrorText := 'Power permit lost';
    AxisData.Diag.udiActualErrorID := 1001;

ELSIF (AxisData.Error.dwLogicalError AND LOG_GLOBAL_DURING_POWER) <> DWORD#0 THEN
    AxisData.Diag.sErrorText := 'Global error during power on';
    AxisData.Diag.udiActualErrorID := 1002;

ELSIF (AxisData.Error.dwLogicalError AND LOG_GLOBAL_DURING_READY) <> DWORD#0 THEN
    AxisData.Diag.sErrorText := 'Global error in READY state';
    AxisData.Diag.udiActualErrorID := 2000;

ELSIF (AxisData.Error.dwLogicalError AND LOG_GLOBAL_DURING_MOTION) <> DWORD#0 THEN
    AxisData.Diag.sErrorText := 'Global error during motion';
    AxisData.Diag.udiActualErrorID := 2100;

ELSIF (AxisData.Error.dwLogicalError AND LOG_JOG_CONFLICT) <> DWORD#0 THEN
    AxisData.Diag.sErrorText := 'Jog positive and negative active together';
    AxisData.Diag.udiActualErrorID := 2001;

ELSIF (AxisData.Error.dwLogicalError AND LOG_MOVE_ABS_NOT_HOMED) <> DWORD#0 THEN
    AxisData.Diag.sErrorText := 'MoveAbsolute denied: axis not homed';
    AxisData.Diag.udiActualErrorID := 1200;

ELSIF (AxisData.Error.dwLogicalError AND LOG_MOVE_REL_NOT_HOMED) <> DWORD#0 THEN
    AxisData.Diag.sErrorText := 'MoveRelative denied: axis not homed';
    AxisData.Diag.udiActualErrorID := 1300;

ELSIF (AxisData.Error.dwLogicalError AND LOG_STEP_TIMEOUT) <> DWORD#0 THEN
    AxisData.Diag.sErrorText := 'Step timeout';
    AxisData.Diag.udiActualErrorID := 9000 + INT_TO_UDINT(AxisData.Diag.iLastErrorStep);

ELSIF (AxisData.Error.dwLogicalError AND LOG_UNKNOWN_STEP) <> DWORD#0 THEN
    AxisData.Diag.sErrorText := 'Unknown axis step';
    AxisData.Diag.udiActualErrorID := 9999;

ELSIF (AxisData.Error.dwAxisError AND AXE_MC_POWER_ERROR) <> DWORD#0 THEN
    AxisData.Diag.sErrorText := 'MC_Power error';
    AxisData.Diag.udiActualErrorID := TO_UDINT(fbPower.ErrorID);

ELSIF (AxisData.Error.dwAxisError AND AXE_MC_RESET_ERROR) <> DWORD#0 THEN
    AxisData.Diag.sErrorText := 'MC_Reset error';
    AxisData.Diag.udiActualErrorID := TO_UDINT(fbReset.ErrorID);

ELSIF (AxisData.Error.dwAxisError AND AXE_MC_STOP_ERROR) <> DWORD#0 THEN
    AxisData.Diag.sErrorText := 'MC_Stop error';
    AxisData.Diag.udiActualErrorID := TO_UDINT(fbStop.ErrorID);

ELSIF (AxisData.Error.dwAxisError AND AXE_MC_JOG_ERROR) <> DWORD#0 THEN
    AxisData.Diag.sErrorText := 'MC_Jog error';
    AxisData.Diag.udiActualErrorID := TO_UDINT(fbJog.ErrorID);

ELSIF (AxisData.Error.dwAxisError AND AXE_MC_HOME_ERROR) <> DWORD#0 THEN
    AxisData.Diag.sErrorText := 'MC_Home error';
    AxisData.Diag.udiActualErrorID := TO_UDINT(fbHome.ErrorID);

ELSIF (AxisData.Error.dwAxisError AND AXE_MC_MOVE_ABS_ERROR) <> DWORD#0 THEN
    AxisData.Diag.sErrorText := 'MC_MoveAbsolute error';
    AxisData.Diag.udiActualErrorID := TO_UDINT(fbMoveAbsolute.ErrorID);

ELSIF (AxisData.Error.dwAxisError AND AXE_MC_MOVE_REL_ERROR) <> DWORD#0 THEN
    AxisData.Diag.sErrorText := 'MC_MoveRelative error';
    AxisData.Diag.udiActualErrorID := TO_UDINT(fbMoveRelative.ErrorID);

ELSIF (AxisData.Error.dwAxisError AND AXE_READ_POS_ERROR) <> DWORD#0 THEN
    AxisData.Diag.sErrorText := 'MC_ReadActualPosition error';
    AxisData.Diag.udiActualErrorID := TO_UDINT(fbReadPosition.ErrorID);

ELSIF (AxisData.Error.dwAxisError AND AXE_READ_STATUS_ERROR) <> DWORD#0 THEN
    AxisData.Diag.sErrorText := 'MC_ReadStatus error';
    AxisData.Diag.udiActualErrorID := TO_UDINT(fbReadStatus.ErrorID);

ELSIF (AxisData.Error.dwAxisError AND AXE_ERRORSTOP) <> DWORD#0 THEN
    AxisData.Diag.sErrorText := 'Axis Errorstop active';
    AxisData.Diag.udiActualErrorID := 3001;

ELSIF (AxisData.Error.dwAxisError AND AXE_FB_ERROR_OCCURRED) <> DWORD#0 THEN
    AxisData.Diag.sErrorText := 'SoftMotion FBErrorOccured active';
    AxisData.Diag.udiActualErrorID := 3002;

ELSIF (AxisData.Error.dwAxisError AND AXE_COMMAND_ABORTED) <> DWORD#0 THEN
    AxisData.Diag.sErrorText := 'Motion command aborted';
    AxisData.Diag.udiActualErrorID := 3003;

ELSIF (AxisData.Error.dwAxisError AND AXE_UNKNOWN_ACTUAL_ERROR) <> DWORD#0 THEN
    AxisData.Diag.sErrorText := 'Unknown actual axis error';
    AxisData.Diag.udiActualErrorID := 3004;

ELSIF (AxisData.Error.dwAxisError AND AXE_DRIVE_AXIS_ERROR) <> DWORD#0 THEN
    AxisData.Diag.sErrorText := 'Drive axis error active';
    AxisData.Diag.udiActualErrorID := DWORD_TO_UDINT(fbReadAxisError.AxisErrorID);

ELSIF AxisData.Command.xGlobalError THEN
    AxisData.Diag.sErrorText := 'Global error active';
    AxisData.Diag.udiActualErrorID := 5000;
END_IF;

IF AxisData.Diag.udiActualErrorID <> 0 THEN
    AxisData.Diag.udiLastErrorID := AxisData.Diag.udiActualErrorID;
END_IF;

// Сохраняем последнюю ненулевую ошибку и формируем удобное представление для HMI.
IF (AxisData.Error.dwAxisError <> DWORD#0)
OR (AxisData.Error.dwLogicalError <> DWORD#0) THEN
	AxisData.Error.dwAxisErrorLast := AxisData.Error.dwAxisError;
	AxisData.Error.dwLogicalErrorLast := AxisData.Error.dwLogicalError;
END_IF;

AxisData.Error.stErrorActive := UpdateErrorView(
	dwAxisError := AxisData.Error.dwAxisError,
	dwLogicalError := AxisData.Error.dwLogicalError
);
AxisData.Error.stErrorLast := UpdateErrorView(
	dwAxisError := AxisData.Error.dwAxisErrorLast,
	dwLogicalError := AxisData.Error.dwLogicalErrorLast
);

(* ---- FB_AXIS_GROUP.st ---- *)
FUNCTION_BLOCK FB_AXIS_GROUP
VAR_INPUT

END_VAR
VAR_OUTPUT
END_VAR
VAR
	// Внутренние исполняемые булевые переменные
	xEnable      : BOOL; // Импульс включения группы
	xRegulatorOn : BOOL; // Запрос включения регуляторов
	xDriveStart  : BOOL; // Запрос разрешения приводов
	xDisable     : BOOL; // Импульс отключения группы
	xPowerEnable : BOOL; // Защёлкнутый запрос питания
	xReset       : BOOL; // Импульс сброса ошибок
	xResetMC     : BOOL; // Выполняется сброс SoftMotion
	xMoveDirect  : BOOL; // Выполняется прямое перемещение
	xMoveLinear  : BOOL; // Выполняется линейное перемещение
	xStopCmd     : BOOL; // Выполняется остановка
	xHaltCmd     : BOOL; // Выполняется плавная остановка

	iPrevStep : E_AXIS_GROUP_STATE; // Предыдущий шаг автомата

	// Для таймера шага
	tonStepTimeout   : TON; // Таймер превышения времени шага
	xStepTimeout     : BOOL; // Время шага превышено
	xStepChanged     : BOOL; // Шаг изменился в текущем цикле
	xStepTimerEnable : BOOL; // Разрешение таймера шага
	xStepInitialized : BOOL; // Предыдущий шаг инициализирован

	// Для удержания предупреждений
    tpWarningHold : TP; // Удержание предупреждения для отображения
    xWarningPulse : BOOL; // Импульс нового предупреждения

	// ФБ группы осей
	fbReadStatus   : MC_GroupReadStatus; // Чтение состояния группы
	fbReadError    : MC_GroupReadError; // Чтение активной ошибки группы
	fbReadPosition : MC_GroupReadActualPosition; // Чтение текущей позиции группы
	fbGroupEnable  : MC_GroupEnable; // Включение группы
	fbGroupDisable : MC_GroupDisable; // Отключение группы
	fbGroupPower   : SMC_GroupPower; // Управление питанием группы
	fbGroupReset   : MC_GroupReset; // Сброс ошибок группы

	fbMoveDirect : MC_MoveDirectAbsolute; // Прямое абсолютное перемещение
	fbMoveLinear : MC_MoveLinearAbsolute; // Линейное абсолютное перемещение

	fbGroupHalt : MC_GroupHalt; // Плавная остановка группы
	fbGroupStop : MC_GroupStop; // Остановка группы

	stPosition : SMC_POS_REF; // Текущая позиция группы

	// Триггеры на команды
    rtEnable        : R_TRIG; // Фронт команды включения
    rtDisable       : R_TRIG; // Фронт команды отключения
	rtEnablePower   : R_TRIG; // Фронт запроса питания
    rtResetAllError : R_TRIG; // Фронт команды сброса
    rtMoveDirect    : R_TRIG; // Фронт прямого перемещения
    rtMoveLinear    : R_TRIG; // Фронт линейного перемещения
	rtStopCmd       : R_TRIG; // Фронт команды остановки
	rtHaltCmd       : R_TRIG; // Фронт плавной остановки

END_VAR
VAR_IN_OUT
	AxisGroup : AXIS_GROUP_REF_SM3; // Ссылка на группу осей SoftMotion
	GroupData : ST_AXIS_GROUP; // Команды, статусы и диагностика группы
END_VAR

VAR CONSTANT
	// ==================================================
    // Логические ошибки группы
    // ==================================================
	LOG_STEP_TIMEOUT             : DWORD := 1; // Превышено время шага
	LOG_INVALID_STATE            : DWORD := 2; // Неизвестный шаг автомата
	LOG_POWER_PERMIT_READY       : DWORD := 4; // Нет разрешения питания в готовности
	LOG_POWER_PERMIT_LOST_DIRECT : DWORD := 8; // Разрешение питания снято при движении
	MASK_LOCAL_LOGICAL_ERROR      : DWORD := LOG_STEP_TIMEOUT OR LOG_INVALID_STATE; // Локальные логические первопричины

	// ==================================================
    // Ошибки блоков движения группы
    // ==================================================
	MOTION_ERR_ENABLE        : DWORD := 1; // Ошибка включения группы
	MOTION_ERR_POWER         : DWORD := 2; // Ошибка питания группы
	MOTION_ERR_DISABLE       : DWORD := 4; // Ошибка отключения группы
	MOTION_ERR_RESET         : DWORD := 8; // Ошибка сброса группы
	MOTION_ERR_MOVE_DIRECT   : DWORD := 16; // Ошибка прямого перемещения
	MOTION_ERR_MOVE_LINEAR   : DWORD := 32; // Ошибка линейного перемещения
	MOTION_ERR_HALT          : DWORD := 64; // Ошибка плавной остановки
	MOTION_ERR_STOP          : DWORD := 128; // Ошибка остановки
	MOTION_ERR_READ_POSITION : DWORD := 256; // Ошибка чтения позиции
	MOTION_ERR_READ_STATUS   : DWORD := 512; // Ошибка чтения статуса
	MOTION_ERR_READ_GROUP_ERROR : DWORD := 1024; // Ошибка чтения кода ошибки группы
	MOTION_ERR_GROUP_ERROR_STOP : DWORD := 2048; // Группа SoftMotion находится в ErrorStop

	WRN_NO_POWER_PERMIT       : UINT := 1; // Нет разрешения питания
	WRN_MOVE_COMMAND_CONFLICT : UINT := 2; // Одновременно заданы два типа движения
	WRN_GLOBAL_ERROR_ACTIVE   : UINT := 3; // Сброс отклонён из-за глобальной ошибки
	WRN_MOTION_ERROR_ACTIVE   : UINT := 4; // Сброс отклонён из-за активной Motion-ошибки
END_VAR

// --- BEGIN IMPLEMENTATION ---

// =============================================================================
// 1. Добить предупреждения и ошибки
// 2. Сделать логирование ошибок и шагов
// 3. Сделать необходимые сигналы статусов
// =============================================================================

// =============================================================================
// 1. Одноцикловые сигналы
// =============================================================================
xWarningPulse := FALSE;

GroupData.Diag.xStepChanged := FALSE;
GroupData.Error.dwLogicalErrorNew := DWORD#0;
GroupData.Error.dwMotionErrorNew := DWORD#0;

// =============================================================================
// 2. Фронты команд
// =============================================================================
rtDisable(CLK := GroupData.Command.xDisable);
rtEnablePower(CLK := GroupData.Command.xPowerEnable);
rtResetAllError(CLK := GroupData.Command.xReset);
rtMoveDirect(CLK := GroupData.Command.xMoveDirect);
rtMoveLinear(CLK := GroupData.Command.xMoveLinear);
rtHaltCmd(CLK := GroupData.Command.xHaltCmd);
rtStopCmd(CLK := GroupData.Command.xStopCmd);

// =============================================================================
// 3. Чтение состояния группы и координат
// =============================================================================
fbReadStatus(
    Enable    := TRUE,
    AxisGroup := AxisGroup
);

fbReadError(
    Enable    := TRUE,
    AxisGroup := AxisGroup
);

fbReadPosition(
    AxisGroup   := AxisGroup,
    Enable      := TRUE,
    CoordSystem := SMC_COORD_SYSTEM.MCS
);

IF fbReadPosition.Valid THEN
    GroupData.Status.ActualX := fbReadPosition.Position.c.X;
    GroupData.Status.ActualY := fbReadPosition.Position.c.Y;
    GroupData.Status.ActualZ := fbReadPosition.Position.c.Z;
END_IF;

// =============================================================================
// 4. Текущий статус ошибок
// =============================================================================
GroupData.Status.xGroupError :=
    fbReadStatus.Error
    OR fbReadStatus.GroupErrorStop
    OR (GroupData.Error.dwMotionErrorLatched <> DWORD#0);

GroupData.Status.xLocalError :=
    GroupData.Status.xGroupError
    OR (GroupData.Error.dwLogicalErrorLatched <> DWORD#0);

// =============================================================================
// 5. Команды Motion FB по умолчанию
// =============================================================================
xEnable := FALSE;
xDisable := FALSE;
xResetMC := FALSE;
xMoveDirect := FALSE;
xMoveLinear := FALSE;
xStopCmd := FALSE;
xHaltCmd := FALSE;

// =============================================================================
// 6. Машина состояний
// =============================================================================
CASE GroupData.Diag.iStep OF

    // -------------------------------------------------------------------------
    E_AXIS_GROUP_STATE.DISABLED:
    // -------------------------------------------------------------------------
        GroupData.Diag.sStepName := 'DISABLED';
        GroupData.Diag.tStepPreset := T#0S;
        GroupData.Diag.iPowerMode := E_AXIS_GROUP_POWER_MODE.OFF;

        IF GroupData.Command.xGlobalError
           OR GroupData.Status.xLocalError THEN

            GroupData.Diag.iStep := E_AXIS_GROUP_STATE.ERROR;

        ELSIF rtEnablePower.Q AND NOT GroupData.Command.xPowerPermit THEN
            GroupData.Diag.sWarningText := 'Power permit is not active';
            GroupData.Diag.stWarning.uiCode := WRN_NO_POWER_PERMIT;
            GroupData.Diag.stWarning.udiSequence := GroupData.Diag.stWarning.udiSequence + UDINT#1;
            IF GroupData.Diag.stWarning.udiSequence = UDINT#0 THEN
                GroupData.Diag.stWarning.udiSequence := UDINT#1;
            END_IF;
            xWarningPulse := TRUE;

        ELSIF rtEnablePower.Q THEN
            GroupData.Diag.iStep := E_AXIS_GROUP_STATE.ENABLING_POWER;
        END_IF;

    // -------------------------------------------------------------------------
    E_AXIS_GROUP_STATE.ENABLING_POWER:
    // -------------------------------------------------------------------------
        GroupData.Diag.sStepName := 'ENABLING_POWER';
        GroupData.Diag.tStepPreset := GroupData.Timeouts.tPowerTimeout;
        GroupData.Diag.iPowerMode := E_AXIS_GROUP_POWER_MODE.ON;

        IF fbReadStatus.GroupErrorStop
           OR fbGroupPower.Error THEN

            GroupData.Diag.iStep := E_AXIS_GROUP_STATE.ERROR;

        ELSIF NOT GroupData.Command.xPowerPermit
           OR GroupData.Command.xGlobalError THEN

            GroupData.Diag.iStep := E_AXIS_GROUP_STATE.DISABLING_POWER;

        ELSIF xStepTimeout THEN
            GroupData.Error.dwLogicalErrorNew :=
                GroupData.Error.dwLogicalErrorNew
                OR LOG_STEP_TIMEOUT;

            GroupData.Diag.iStep := E_AXIS_GROUP_STATE.DISABLING_POWER;

        ELSIF fbGroupPower.Status THEN
            GroupData.Diag.iStep := E_AXIS_GROUP_STATE.ENABLING_GROUP;
        END_IF;

    // -------------------------------------------------------------------------
    E_AXIS_GROUP_STATE.ENABLING_GROUP:
    // -------------------------------------------------------------------------
        GroupData.Diag.sStepName := 'ENABLING_GROUP';
        GroupData.Diag.tStepPreset := GroupData.Timeouts.tGroupTimeout;
        GroupData.Diag.iPowerMode := E_AXIS_GROUP_POWER_MODE.ON;

        xEnable := TRUE;

        IF fbReadStatus.GroupErrorStop
           OR fbGroupEnable.Error THEN

            GroupData.Diag.iStep := E_AXIS_GROUP_STATE.ERROR;

        ELSIF NOT GroupData.Command.xPowerPermit
           OR GroupData.Command.xGlobalError THEN

            GroupData.Diag.iStep := E_AXIS_GROUP_STATE.DISABLING_GROUP;

        ELSIF xStepTimeout THEN
            GroupData.Error.dwLogicalErrorNew :=
                GroupData.Error.dwLogicalErrorNew
                OR LOG_STEP_TIMEOUT;

            GroupData.Diag.iStep := E_AXIS_GROUP_STATE.DISABLING_GROUP;

        ELSIF fbGroupEnable.Done
           AND fbReadStatus.GroupStandby THEN

            GroupData.Diag.iStep := E_AXIS_GROUP_STATE.READY;
        END_IF;

    // -------------------------------------------------------------------------
    E_AXIS_GROUP_STATE.READY:
    // -------------------------------------------------------------------------
        GroupData.Diag.sStepName := 'READY';
        GroupData.Diag.tStepPreset := T#0S;
        GroupData.Diag.iPowerMode := E_AXIS_GROUP_POWER_MODE.ON;

        xEnable := TRUE;

        IF fbReadStatus.GroupErrorStop THEN
            GroupData.Diag.iStep := E_AXIS_GROUP_STATE.ERROR;

        ELSIF NOT GroupData.Command.xPowerPermit
           OR GroupData.Command.xGlobalError
           OR GroupData.Status.xLocalError
           OR rtDisable.Q THEN

            GroupData.Diag.iStep := E_AXIS_GROUP_STATE.DISABLING_GROUP;

        ELSIF rtMoveDirect.Q AND rtMoveLinear.Q THEN
            GroupData.Diag.sWarningText :=
                'MoveDirect and MoveLinear requested together';

            GroupData.Diag.stWarning.uiCode := WRN_MOVE_COMMAND_CONFLICT;
            GroupData.Diag.stWarning.udiSequence := GroupData.Diag.stWarning.udiSequence + UDINT#1;
            IF GroupData.Diag.stWarning.udiSequence = UDINT#0 THEN
                GroupData.Diag.stWarning.udiSequence := UDINT#1;
            END_IF;

            xWarningPulse := TRUE;

        ELSIF rtMoveDirect.Q THEN
            GroupData.Diag.iStep := E_AXIS_GROUP_STATE.MOVING_DIRECT;

        ELSIF rtMoveLinear.Q THEN
            GroupData.Diag.iStep := E_AXIS_GROUP_STATE.MOVING_LINEAR;
        END_IF;

    // -------------------------------------------------------------------------
    E_AXIS_GROUP_STATE.MOVING_DIRECT:
    // -------------------------------------------------------------------------
        GroupData.Diag.sStepName := 'MOVING_DIRECT';
        GroupData.Diag.tStepPreset := GroupData.Timeouts.tMoveTimeout;
        GroupData.Diag.iPowerMode := E_AXIS_GROUP_POWER_MODE.ON;

        xEnable := TRUE;
        xMoveDirect := TRUE;

        IF fbReadStatus.GroupErrorStop THEN
            GroupData.Diag.iStep := E_AXIS_GROUP_STATE.ERROR;

        ELSIF fbMoveDirect.Error THEN
            IF fbReadStatus.GroupMoving THEN
                GroupData.Diag.iStep := E_AXIS_GROUP_STATE.EMG_STOP;
            ELSE
                GroupData.Diag.iStep := E_AXIS_GROUP_STATE.ERROR;
            END_IF;

        ELSIF xStepTimeout THEN
            GroupData.Error.dwLogicalErrorNew :=
                GroupData.Error.dwLogicalErrorNew
                OR LOG_STEP_TIMEOUT;

            GroupData.Diag.iStep := E_AXIS_GROUP_STATE.EMG_STOP;

        ELSIF NOT GroupData.Command.xPowerPermit
           OR GroupData.Command.xGlobalError
           OR GroupData.Status.xLocalError
           OR rtStopCmd.Q THEN

            GroupData.Diag.iStep := E_AXIS_GROUP_STATE.EMG_STOP;

        ELSIF rtHaltCmd.Q THEN
            GroupData.Diag.iStep := E_AXIS_GROUP_STATE.HALT_STOP;

        ELSIF fbMoveDirect.Done
           AND fbReadStatus.GroupStandby THEN

            GroupData.Diag.iStep := E_AXIS_GROUP_STATE.READY;
        END_IF;

    // -------------------------------------------------------------------------
    E_AXIS_GROUP_STATE.HALT_STOP:
    // -------------------------------------------------------------------------
        GroupData.Diag.sStepName := 'HALT_STOP';
        GroupData.Diag.tStepPreset := GroupData.Timeouts.tHaltTimeout;
        GroupData.Diag.iPowerMode := E_AXIS_GROUP_POWER_MODE.ON;

        xEnable := TRUE;
        xHaltCmd := TRUE;

        IF fbReadStatus.GroupErrorStop THEN
            GroupData.Diag.iStep := E_AXIS_GROUP_STATE.ERROR;

        ELSIF fbGroupHalt.Error
           OR xStepTimeout
           OR NOT GroupData.Command.xPowerPermit
           OR GroupData.Command.xGlobalError
           OR GroupData.Status.xLocalError
           OR rtStopCmd.Q THEN

            IF xStepTimeout THEN
                GroupData.Error.dwLogicalErrorNew :=
                    GroupData.Error.dwLogicalErrorNew
                    OR LOG_STEP_TIMEOUT;
            END_IF;

            GroupData.Diag.iStep := E_AXIS_GROUP_STATE.EMG_STOP;

        ELSIF fbGroupHalt.Done
           AND fbReadStatus.GroupStandby THEN

            GroupData.Diag.iStep := E_AXIS_GROUP_STATE.READY;
        END_IF;

    // -------------------------------------------------------------------------
    E_AXIS_GROUP_STATE.EMG_STOP:
    // -------------------------------------------------------------------------
        GroupData.Diag.sStepName := 'STOPPING';
        GroupData.Diag.tStepPreset := GroupData.Timeouts.tStopTimeout;
        GroupData.Diag.iPowerMode := E_AXIS_GROUP_POWER_MODE.ON;

        xEnable := TRUE;
        xStopCmd := TRUE;

        IF fbReadStatus.GroupErrorStop
           OR fbGroupStop.Error THEN

            GroupData.Diag.iStep := E_AXIS_GROUP_STATE.ERROR;

        ELSIF xStepTimeout THEN
            GroupData.Error.dwLogicalErrorNew :=
                GroupData.Error.dwLogicalErrorNew
                OR LOG_STEP_TIMEOUT;

            GroupData.Diag.iStep := E_AXIS_GROUP_STATE.ERROR;

        ELSIF fbGroupStop.Done THEN
            GroupData.Diag.iStep := E_AXIS_GROUP_STATE.WAIT_STOP;
        END_IF;

    // -------------------------------------------------------------------------
    E_AXIS_GROUP_STATE.WAIT_STOP:
    // -------------------------------------------------------------------------
        GroupData.Diag.sStepName := 'WAIT_STOP';
        GroupData.Diag.tStepPreset := GroupData.Timeouts.tStopTimeout;
        GroupData.Diag.iPowerMode := E_AXIS_GROUP_POWER_MODE.ON;

        xEnable := TRUE;

        IF fbReadStatus.GroupErrorStop THEN
            GroupData.Diag.iStep := E_AXIS_GROUP_STATE.ERROR;

        ELSIF xStepTimeout THEN
            GroupData.Error.dwLogicalErrorNew :=
                GroupData.Error.dwLogicalErrorNew
                OR LOG_STEP_TIMEOUT;

            GroupData.Diag.iStep := E_AXIS_GROUP_STATE.ERROR;

        ELSIF fbReadStatus.GroupStandby THEN
            GroupData.Diag.iStep := E_AXIS_GROUP_STATE.DISABLING_GROUP;
        END_IF;

    // -------------------------------------------------------------------------
    E_AXIS_GROUP_STATE.DISABLING_GROUP:
    // -------------------------------------------------------------------------
        GroupData.Diag.sStepName := 'DISABLING_GROUP';
        GroupData.Diag.tStepPreset := GroupData.Timeouts.tGroupTimeout;
        GroupData.Diag.iPowerMode := E_AXIS_GROUP_POWER_MODE.ON;

        xDisable := TRUE;

        IF fbReadStatus.GroupErrorStop
           OR fbGroupDisable.Error THEN

            GroupData.Diag.iStep := E_AXIS_GROUP_STATE.ERROR;

        ELSIF xStepTimeout THEN
            GroupData.Error.dwLogicalErrorNew :=
                GroupData.Error.dwLogicalErrorNew
                OR LOG_STEP_TIMEOUT;

            GroupData.Diag.iStep := E_AXIS_GROUP_STATE.ERROR;

        ELSIF fbGroupDisable.Done
           AND fbReadStatus.GroupDisabled THEN

            GroupData.Diag.iStep := E_AXIS_GROUP_STATE.DISABLING_POWER;
        END_IF;

    // -------------------------------------------------------------------------
    E_AXIS_GROUP_STATE.DISABLING_POWER:
    // -------------------------------------------------------------------------
        GroupData.Diag.sStepName := 'DISABLING_POWER';
        GroupData.Diag.tStepPreset := GroupData.Timeouts.tPowerTimeout;
        GroupData.Diag.iPowerMode :=
            E_AXIS_GROUP_POWER_MODE.OFF_REQUEST;

        IF xStepTimeout THEN
            GroupData.Error.dwLogicalErrorNew :=
                GroupData.Error.dwLogicalErrorNew
                OR LOG_STEP_TIMEOUT;

            GroupData.Diag.iStep := E_AXIS_GROUP_STATE.ERROR;

        ELSIF NOT fbGroupPower.Status THEN

            IF GroupData.Command.xGlobalError
               OR GroupData.Status.xLocalError
			   OR NOT GroupData.Command.xPowerPermit THEN

                GroupData.Diag.iStep := E_AXIS_GROUP_STATE.ERROR;
            ELSE
                GroupData.Diag.iStep := E_AXIS_GROUP_STATE.DISABLED;
            END_IF;
        END_IF;

    // -------------------------------------------------------------------------
    E_AXIS_GROUP_STATE.ERROR:
    // -------------------------------------------------------------------------
        GroupData.Diag.sStepName := 'ERROR';
        GroupData.Diag.tStepPreset := T#0S;

        GroupData.Diag.iPowerMode := E_AXIS_GROUP_POWER_MODE.OFF_REQUEST;

        IF rtResetAllError.Q THEN

            IF GroupData.Command.xGlobalError THEN
                GroupData.Diag.sWarningText :=
                    'Global error is still active';

                GroupData.Diag.stWarning.uiCode := WRN_GLOBAL_ERROR_ACTIVE;
                GroupData.Diag.stWarning.udiSequence := GroupData.Diag.stWarning.udiSequence + UDINT#1;
                IF GroupData.Diag.stWarning.udiSequence = UDINT#0 THEN
                    GroupData.Diag.stWarning.udiSequence := UDINT#1;
                END_IF;

                xWarningPulse := TRUE;

            ELSIF fbReadStatus.GroupErrorStop THEN
                    GroupData.Diag.iStep :=
                        E_AXIS_GROUP_STATE.RESETTING;

            ELSIF GroupData.Error.dwMotionErrorActive
                  <> DWORD#0 THEN

                GroupData.Diag.sWarningText :=
                    'Motion FB error is still active';

                GroupData.Diag.stWarning.uiCode := WRN_MOTION_ERROR_ACTIVE;
                GroupData.Diag.stWarning.udiSequence := GroupData.Diag.stWarning.udiSequence + UDINT#1;
                IF GroupData.Diag.stWarning.udiSequence = UDINT#0 THEN
                    GroupData.Diag.stWarning.udiSequence := UDINT#1;
                END_IF;

                xWarningPulse := TRUE;

            ELSE
                // Ошибка устранена — очищаем защёлки.
                GroupData.Error.dwLogicalErrorLatched := DWORD#0;
                GroupData.Error.dwMotionErrorLatched := DWORD#0;
                GroupData.Error.dwMotionErrorPrevious := DWORD#0;

                IF NOT fbGroupPower.Status THEN
                    GroupData.Diag.iStep :=
                        E_AXIS_GROUP_STATE.DISABLED;

                ELSIF fbReadStatus.GroupDisabled THEN
                    GroupData.Diag.iStep :=
                        E_AXIS_GROUP_STATE.DISABLING_POWER;

                ELSIF fbReadStatus.GroupStandby THEN
                    GroupData.Diag.iStep :=
                        E_AXIS_GROUP_STATE.DISABLING_GROUP;

                ELSE
                    GroupData.Diag.iStep :=
                        E_AXIS_GROUP_STATE.DISABLING_POWER;
                END_IF;
            END_IF;
        END_IF;

    // -------------------------------------------------------------------------
    E_AXIS_GROUP_STATE.RESETTING:
    // -------------------------------------------------------------------------
        GroupData.Diag.sStepName := 'RESETTING';
        GroupData.Diag.tStepPreset := GroupData.Timeouts.tGroupTimeout;
        GroupData.Diag.iPowerMode := E_AXIS_GROUP_POWER_MODE.ON;

        xResetMC := TRUE;

        IF GroupData.Command.xGlobalError
           OR fbGroupReset.Error THEN

            GroupData.Diag.iStep := E_AXIS_GROUP_STATE.ERROR;

        ELSIF xStepTimeout THEN
            GroupData.Error.dwLogicalErrorNew :=
                GroupData.Error.dwLogicalErrorNew
                OR LOG_STEP_TIMEOUT;

            GroupData.Diag.iStep := E_AXIS_GROUP_STATE.ERROR;

        ELSIF fbGroupReset.Done THEN
            // Статус группы был прочитан до вызова MC_GroupReset.
            // Проверяем результат сброса только со следующего цикла.
            GroupData.Diag.iStep := E_AXIS_GROUP_STATE.RESET_VERIFY;
        END_IF;

    // -------------------------------------------------------------------------
    E_AXIS_GROUP_STATE.RESET_VERIFY:
    // -------------------------------------------------------------------------
        GroupData.Diag.sStepName := 'RESET_VERIFY';
        GroupData.Diag.tStepPreset := GroupData.Timeouts.tGroupTimeout;
        GroupData.Diag.iPowerMode := E_AXIS_GROUP_POWER_MODE.ON;

        IF GroupData.Command.xGlobalError THEN
            GroupData.Diag.iStep := E_AXIS_GROUP_STATE.ERROR;

        ELSIF xStepTimeout THEN
            GroupData.Error.dwLogicalErrorNew :=
                GroupData.Error.dwLogicalErrorNew
                OR LOG_STEP_TIMEOUT;

            GroupData.Diag.iStep := E_AXIS_GROUP_STATE.ERROR;

        ELSIF fbReadStatus.Valid
           AND fbReadStatus.GroupErrorStop
           AND fbReadError.Valid
           AND (TO_UDINT(fbReadError.GroupErrorID) <> UDINT#0) THEN

            // Причина ошибки осталась активной после завершения сброса.
            GroupData.Diag.iStep := E_AXIS_GROUP_STATE.ERROR;

        ELSIF fbReadStatus.Valid
           AND NOT fbReadStatus.GroupErrorStop THEN

            GroupData.Error.dwLogicalErrorLatched := DWORD#0;
            GroupData.Error.dwMotionErrorLatched := DWORD#0;
            GroupData.Error.dwMotionErrorPrevious := DWORD#0;

            IF NOT fbGroupPower.Status THEN
                GroupData.Diag.iStep := E_AXIS_GROUP_STATE.DISABLED;

            ELSIF fbReadStatus.GroupDisabled THEN
                GroupData.Diag.iStep := E_AXIS_GROUP_STATE.DISABLING_POWER;

            ELSIF fbReadStatus.GroupStandby THEN
                GroupData.Diag.iStep := E_AXIS_GROUP_STATE.DISABLING_GROUP;

            ELSE
                GroupData.Diag.iStep := E_AXIS_GROUP_STATE.DISABLING_POWER;
            END_IF;
        END_IF;

    // -------------------------------------------------------------------------
    ELSE
    // -------------------------------------------------------------------------
        GroupData.Error.dwLogicalErrorNew :=
            GroupData.Error.dwLogicalErrorNew
            OR LOG_INVALID_STATE;

        GroupData.Diag.iStep := E_AXIS_GROUP_STATE.ERROR;

END_CASE;

// =============================================================================
// 7. Целевая позиция
// =============================================================================
GroupData.MotionParam.stTargetPos.c.X := GroupData.MotionParam.lrX;
GroupData.MotionParam.stTargetPos.c.Y := GroupData.MotionParam.lrY;
GroupData.MotionParam.stTargetPos.c.Z := GroupData.MotionParam.lrZ;

// =============================================================================
// 8. Режим питания
// =============================================================================
xPowerEnable :=
    GroupData.Diag.iPowerMode <> E_AXIS_GROUP_POWER_MODE.OFF;

xRegulatorOn :=
    GroupData.Diag.iPowerMode = E_AXIS_GROUP_POWER_MODE.ON;

xDriveStart :=
    GroupData.Diag.iPowerMode = E_AXIS_GROUP_POWER_MODE.ON;

// =============================================================================
// 9. Вызовы Motion FB
// =============================================================================
fbGroupEnable(
    AxisGroup := AxisGroup,
    Execute   := xEnable
);

fbGroupDisable(
    AxisGroup := AxisGroup,
    Execute   := xDisable
);

fbGroupPower(
    AxisGroup    := AxisGroup,
    Enable       := xPowerEnable,
    bRegulatorOn := xRegulatorOn,
    bDriveStart  := xDriveStart
);

fbGroupReset(
    AxisGroup := AxisGroup,
    Execute   := xResetMC
);

fbMoveDirect(
    AxisGroup   := AxisGroup,
    Execute     := xMoveDirect,
    Position    := GroupData.MotionParam.stTargetPos,
    CoordSystem := SMC_COORD_SYSTEM.MCS,
    BufferMode  := MC_BUFFER_MODE.Aborting,
    VelFactor   := GroupData.MotionParam.VelFactor,
    AccFactor   := GroupData.MotionParam.AccFactor,
    JerkFactor  := GroupData.MotionParam.JerkFactor
);

fbMoveLinear(
    AxisGroup := AxisGroup,
    Execute   := xMoveLinear
);

fbGroupHalt(
    AxisGroup    := AxisGroup,
    Execute      := xHaltCmd,
    Deceleration := GroupData.MotionParam.HaltDeceleration,
    Jerk         := GroupData.MotionParam.HaltJerk
);

fbGroupStop(
    AxisGroup    := AxisGroup,
    Execute      := xStopCmd,
    Deceleration := GroupData.MotionParam.HaltDeceleration * 2,
    Jerk         := GroupData.MotionParam.HaltJerk * 2
);

// =============================================================================
// 10. Маска Motion-ошибок
// =============================================================================
GroupData.Error.dwMotionErrorActive := DWORD#0;

IF fbGroupEnable.Error THEN
    GroupData.Error.dwMotionErrorActive :=
        GroupData.Error.dwMotionErrorActive
        OR MOTION_ERR_ENABLE;
END_IF;

IF fbGroupPower.Error THEN
    GroupData.Error.dwMotionErrorActive :=
        GroupData.Error.dwMotionErrorActive
        OR MOTION_ERR_POWER;
END_IF;

IF fbGroupDisable.Error THEN
    GroupData.Error.dwMotionErrorActive :=
        GroupData.Error.dwMotionErrorActive
        OR MOTION_ERR_DISABLE;
END_IF;

IF fbGroupReset.Error THEN
    GroupData.Error.dwMotionErrorActive :=
        GroupData.Error.dwMotionErrorActive
        OR MOTION_ERR_RESET;
END_IF;

IF fbMoveDirect.Error THEN
    GroupData.Error.dwMotionErrorActive :=
        GroupData.Error.dwMotionErrorActive
        OR MOTION_ERR_MOVE_DIRECT;
END_IF;

IF fbMoveLinear.Error THEN
    GroupData.Error.dwMotionErrorActive :=
        GroupData.Error.dwMotionErrorActive
        OR MOTION_ERR_MOVE_LINEAR;
END_IF;

IF fbGroupHalt.Error THEN
    GroupData.Error.dwMotionErrorActive :=
        GroupData.Error.dwMotionErrorActive
        OR MOTION_ERR_HALT;
END_IF;

IF fbGroupStop.Error THEN
    GroupData.Error.dwMotionErrorActive :=
        GroupData.Error.dwMotionErrorActive
        OR MOTION_ERR_STOP;
END_IF;

IF fbReadPosition.Error THEN
    GroupData.Error.dwMotionErrorActive :=
        GroupData.Error.dwMotionErrorActive
        OR MOTION_ERR_READ_POSITION;
END_IF;

IF fbReadStatus.Error THEN
    GroupData.Error.dwMotionErrorActive :=
        GroupData.Error.dwMotionErrorActive
        OR MOTION_ERR_READ_STATUS;
END_IF;

IF fbReadError.Error THEN
    GroupData.Error.dwMotionErrorActive :=
        GroupData.Error.dwMotionErrorActive
        OR MOTION_ERR_READ_GROUP_ERROR;
END_IF;

IF fbReadStatus.GroupErrorStop THEN
    GroupData.Error.dwMotionErrorActive :=
        GroupData.Error.dwMotionErrorActive
        OR MOTION_ERR_GROUP_ERROR_STOP;
END_IF;

// Только ошибки, которых не было в предыдущем цикле.
GroupData.Error.dwMotionErrorNew :=
    GroupData.Error.dwMotionErrorActive
    AND NOT GroupData.Error.dwMotionErrorPrevious;

// Защёлкиваем новые логические и Motion-ошибки.
GroupData.Error.dwLogicalErrorLatched :=
    GroupData.Error.dwLogicalErrorLatched
    OR GroupData.Error.dwLogicalErrorNew;

GroupData.Error.dwMotionErrorLatched :=
    GroupData.Error.dwMotionErrorLatched
    OR GroupData.Error.dwMotionErrorNew;

// Сохраняем Motion-маску для следующего цикла.
GroupData.Error.dwMotionErrorPrevious :=
    GroupData.Error.dwMotionErrorActive;

GroupData.Error.dwAlarmActive :=
    GroupData.Error.dwMotionErrorLatched
    OR SHL(GroupData.Error.dwLogicalErrorLatched AND MASK_LOCAL_LOGICAL_ERROR, 16);

// =============================================================================
// 11. Изменение шага и таймер
// =============================================================================
IF NOT xStepInitialized THEN
    iPrevStep := GroupData.Diag.iStep;
    xStepInitialized := TRUE;
END_IF;

xStepChanged :=
    GroupData.Diag.iStep <> iPrevStep;

GroupData.Diag.xStepChanged := xStepChanged;

IF xStepChanged THEN
    GroupData.Diag.iOldStep := iPrevStep;
    GroupData.Diag.iNewStep := GroupData.Diag.iStep;
    iPrevStep := GroupData.Diag.iStep;
END_IF;

// При переходе в новый шаг таймер один цикл выключен.
// Со следующего цикла начинается отсчёт нового шага.
tonStepTimeout(
    IN :=
        NOT xStepChanged
        AND (GroupData.Diag.tStepPreset > T#0S)
        AND (GroupData.Diag.iStep <> E_AXIS_GROUP_STATE.ERROR),

    PT := GroupData.Diag.tStepPreset
);

xStepTimeout := tonStepTimeout.Q;
GroupData.Diag.xStepTimeout := xStepTimeout;

// =============================================================================
// 12. Финальные статусы
// =============================================================================
GroupData.Status.xGroupError :=
    fbReadStatus.Error
    OR fbReadStatus.GroupErrorStop
    OR (GroupData.Error.dwMotionErrorLatched <> DWORD#0);

GroupData.Status.xLocalError :=
    GroupData.Status.xGroupError
    OR (GroupData.Error.dwLogicalErrorLatched <> DWORD#0);

GroupData.Status.xMoveDirectDone := fbMoveDirect.Done;

// Код ошибки самой группы не совпадает с ErrorID диагностических Motion FB.
IF fbReadError.Valid
   AND (TO_UDINT(fbReadError.GroupErrorID) <> UDINT#0) THEN
    GroupData.Diag.udiActualErrorID := TO_UDINT(fbReadError.GroupErrorID);
    GroupData.Diag.sErrorText := 'Axis group error';
ELSIF fbGroupReset.Error THEN
    GroupData.Diag.udiActualErrorID := TO_UDINT(fbGroupReset.ErrorID);
    GroupData.Diag.sErrorText := 'MC_GroupReset error';
ELSE
    GroupData.Diag.udiActualErrorID := UDINT#0;
    GroupData.Diag.sErrorText := '';
END_IF;

IF GroupData.Diag.udiActualErrorID <> UDINT#0 THEN
    GroupData.Diag.udiLastErrorID := GroupData.Diag.udiActualErrorID;
END_IF;

// Сохраняем последнюю ненулевую ошибку и формируем удобное представление для HMI.
IF (GroupData.Error.dwMotionErrorLatched <> DWORD#0)
OR (GroupData.Error.dwLogicalErrorLatched <> DWORD#0) THEN
	GroupData.Error.dwMotionErrorLast := GroupData.Error.dwMotionErrorLatched;
	GroupData.Error.dwLogicalErrorLast := GroupData.Error.dwLogicalErrorLatched;
END_IF;

GroupData.Error.stErrorActive := UpdateErrorView(
	dwMotionError := GroupData.Error.dwMotionErrorLatched OR GroupData.Error.dwMotionErrorActive,
	dwLogicalError := GroupData.Error.dwLogicalErrorLatched
);
GroupData.Error.stErrorLast := UpdateErrorView(
	dwMotionError := GroupData.Error.dwMotionErrorLast,
	dwLogicalError := GroupData.Error.dwLogicalErrorLast
);

(* ---- FB_CELL_MANAGER.st ---- *)
FUNCTION_BLOCK FB_CELL_MANAGER
VAR_INPUT
	xStart            : BOOL; // Импульс запуска автоматического цикла
	xStop             : BOOL; // Импульс остановки автоматического цикла
	xReset            : BOOL; // Сброс ошибок менеджера ячейки
	xManual           : BOOL; // Ручной режим ячейки
	xGlobalError      : BOOL; // Глобальная ошибка ячейки
	xDrivesReady      : BOOL; // Приводы и группа осей готовы к движению
	stRobotStatus     : ST_ROBOT_STATUS; // Состояние робота
	stMagazineStatus  : ST_MAGAZINE_STATUS; // Состояние магазина
	astMachineStatus  : ARRAY [1..3] OF ST_MACHINE_PUBLIC; // Состояния станков
	astMachineDiag    : ARRAY [1..3] OF ST_MACHINE_DIAG; // Состояния автоматов станков
END_VAR
VAR_OUTPUT
	Command : ST_CELL_COMMAND; // Команды оборудованию ячейки
	Status  : ST_CELL_STATUS; // Рабочие статусы ячейки
	Diag    : ST_CELL_DIAG; // Состояние автомата ячейки
	Error   : ST_CELL_ERRORS; // Активные и последние ошибки
END_VAR
VAR
	rtStart            : R_TRIG; // Фронт запуска автоматического цикла
	rtStop             : R_TRIG; // Фронт остановки автоматического цикла
	rtReset            : R_TRIG; // Фронт общего сброса ошибок ячейки
	xRunning           : BOOL; // Защёлка запущенного автоматического цикла
	xStopRequested     : BOOL; // Запрос остановки после безопасного шага
	xCandidateFound    : BOOL; // Найден подходящий станок
	xTimedCandidate    : BOOL; // Найден станок с оценкой оставшегося времени
	uiSelectedMachine  : UINT; // Номер выбранного станка
	uiLoop             : UINT; // Индекс поиска станка
	uiReadyMachines    : UINT; // Количество станков, готовых к работе ячейки
	tMinimumRemaining  : TIME; // Минимальное оставшееся время
	eMagazineOperation : E_MAGAZINE_OPERATION; // Операция магазина текущего шага
	xRobotReady        : BOOL; // Робот готов принять команду
	xMagazineReady     : BOOL; // Магазин готов принять команду
	xReadyToStart      : BOOL; // Выполнены все условия запуска автоматического цикла
END_VAR
VAR CONSTANT
	ERR_BOTH_GRIPPERS : DWORD := DWORD#16#0000_0001; // Одновременно заняты оба захвата
	ERR_ROBOT         : DWORD := DWORD#16#0000_0002; // Ошибка робота
	ERR_MAGAZINE      : DWORD := DWORD#16#0000_0004; // Ошибка магазина
	ERR_MACHINE       : DWORD := DWORD#16#0000_0008; // Ошибка станка во время обслуживания
	ERR_GLOBAL_STOP   : DWORD := DWORD#16#0000_0010; // Глобальная ошибка ячейки
	WRN_RESET_GLOBAL_ERROR  : UINT := 1; // Сброс отклонён из-за глобальной ошибки
	WRN_RESET_ROBOT_ERROR   : UINT := 2; // Сброс отклонён из-за ошибки робота
	WRN_RESET_MAGAZINE_ERROR: UINT := 3; // Сброс отклонён из-за ошибки магазина
END_VAR

// --- BEGIN IMPLEMENTATION ---

rtStart(CLK := xStart);
rtStop(CLK := xStop);
rtReset(CLK := xReset);

// Менеджер ячейки предупреждает только о причинах отказа общего сброса.
IF rtReset.Q
AND (Diag.eState = E_CELL_STATE.ERROR) THEN
	IF xGlobalError THEN
		Diag.stWarning.uiCode := WRN_RESET_GLOBAL_ERROR;
	ELSIF stRobotStatus.xError THEN
		Diag.stWarning.uiCode := WRN_RESET_ROBOT_ERROR;
	ELSIF stMagazineStatus.xError THEN
		Diag.stWarning.uiCode := WRN_RESET_MAGAZINE_ERROR;
	ELSE
		Diag.stWarning.uiCode := UINT#0;
	END_IF;

	IF Diag.stWarning.uiCode <> UINT#0 THEN
		Diag.stWarning.udiSequence := Diag.stWarning.udiSequence + UDINT#1;
		IF Diag.stWarning.udiSequence = UDINT#0 THEN
			Diag.stWarning.udiSequence := UDINT#1;
		END_IF;
	END_IF;
END_IF;

IF rtStop.Q OR xManual THEN
	xStopRequested := TRUE;
END_IF;

// Команды по умолчанию снимаются после каждого шага.
Command.stRobot.xExecute := FALSE;
Command.stRobot.xStop := FALSE;
Command.stRobot.xReset := xReset;
Command.stRobot.eAction := E_ROBOT_ACTION.NONE;
Command.stRobot.eSetPoint := E_POINT_NAME.NONE;
Command.stRobot.iTakeSlot := 0;
Command.stRobot.iPutSlot := 0;

Command.stMagazine.xEnable := FALSE;
Command.stMagazine.xDisable := FALSE;
Command.stMagazine.xExecute := FALSE;
Command.stMagazine.xStop := FALSE;

FOR uiLoop := 1 TO 3 DO
	Command.axMachineExecute[uiLoop] := FALSE;
END_FOR;

// Готовность запуска формируется в одном месте и передаётся в HMI.
uiReadyMachines := 0;

FOR uiLoop := 1 TO 3 DO
	IF astMachineStatus[uiLoop].xEnabled
	AND NOT astMachineStatus[uiLoop].xError
	AND (astMachineDiag[uiLoop].eState = E_MACHINE_STATE.IDLE) THEN
		uiReadyMachines := uiReadyMachines + 1;
	END_IF;
END_FOR;

xRobotReady := NOT stRobotStatus.xBusy
	AND NOT stRobotStatus.xError
	AND NOT (stRobotStatus.xBlankAvailable AND stRobotStatus.xDetailAvailable);

xMagazineReady := stMagazineStatus.xEnabled
	AND stMagazineStatus.xReady
	AND stMagazineStatus.xCanEnable
	AND NOT stMagazineStatus.xBusy
	AND NOT stMagazineStatus.xError
	AND NOT stMagazineStatus.xDisablePending
	AND NOT stMagazineStatus.xFinished;

xReadyToStart := (Diag.eState = E_CELL_STATE.IDLE)
	AND NOT xRunning
	AND NOT xManual
	AND NOT xGlobalError
	AND (Error.dwErrorActive = DWORD#0)
	AND xDrivesReady
	AND xRobotReady
	AND xMagazineReady
	AND (uiReadyMachines > 0);

// В состояниях ожидания автомат можно остановить сразу.
IF xStopRequested
AND ((Diag.eState = E_CELL_STATE.ROUTE_PAYLOAD)
	OR (Diag.eState = E_CELL_STATE.SELECT_MACHINE)
	OR (Diag.eState = E_CELL_STATE.WAIT_MACHINE)
	OR (Diag.eState = E_CELL_STATE.WAIT_MAGAZINE)) THEN
	xRunning := FALSE;
	uiSelectedMachine := 0;
	eMagazineOperation := E_MAGAZINE_OPERATION.NONE;
	Diag.eState := E_CELL_STATE.IDLE;
END_IF;

IF xGlobalError
AND (Diag.eState <> E_CELL_STATE.IDLE)
AND (Diag.eState <> E_CELL_STATE.ERROR) THEN
	Error.dwErrorActive := Error.dwErrorActive OR ERR_GLOBAL_STOP;
	Diag.eState := E_CELL_STATE.ERROR;
END_IF;

CASE Diag.eState OF
	E_CELL_STATE.IDLE:
		xRunning := FALSE;
		xStopRequested := FALSE;
		uiSelectedMachine := 0;
		eMagazineOperation := E_MAGAZINE_OPERATION.NONE;

		IF rtStart.Q
		AND xReadyToStart THEN
			xRunning := TRUE;
			Diag.eState := E_CELL_STATE.ROUTE_PAYLOAD;
		END_IF;

	E_CELL_STATE.ROUTE_PAYLOAD:
		uiSelectedMachine := 0;
		eMagazineOperation := E_MAGAZINE_OPERATION.NONE;

		IF stRobotStatus.xError THEN
			Error.dwErrorActive := Error.dwErrorActive OR ERR_ROBOT;
			Diag.eState := E_CELL_STATE.ERROR;

		ELSIF stRobotStatus.xBlankAvailable
		AND stRobotStatus.xDetailAvailable THEN
			Error.dwErrorActive := Error.dwErrorActive OR ERR_BOTH_GRIPPERS;
			Diag.eState := E_CELL_STATE.ERROR;

		ELSIF stRobotStatus.xBlankAvailable THEN
			Diag.eState := E_CELL_STATE.SELECT_MACHINE;

		ELSIF stRobotStatus.xDetailAvailable THEN
			IF stMagazineStatus.xError THEN
				Error.dwErrorActive := Error.dwErrorActive OR ERR_MAGAZINE;
				Diag.eState := E_CELL_STATE.ERROR;
			ELSIF NOT stMagazineStatus.xEnabled THEN
				Diag.eState := E_CELL_STATE.WAIT_MAGAZINE;
			ELSIF stMagazineStatus.xCanChange THEN
				eMagazineOperation := E_MAGAZINE_OPERATION.CHANGE;
				Diag.eState := E_CELL_STATE.MAGAZINE;
			ELSIF stMagazineStatus.xCanPut THEN
				eMagazineOperation := E_MAGAZINE_OPERATION.PUT;
				Diag.eState := E_CELL_STATE.MAGAZINE;
			ELSE
				Diag.eState := E_CELL_STATE.WAIT_MAGAZINE;
			END_IF;

		ELSE
			IF stMagazineStatus.xError THEN
				Error.dwErrorActive := Error.dwErrorActive OR ERR_MAGAZINE;
				Diag.eState := E_CELL_STATE.ERROR;
			ELSIF NOT stMagazineStatus.xEnabled THEN
				Diag.eState := E_CELL_STATE.WAIT_MAGAZINE;
			ELSIF stMagazineStatus.xCanTake THEN
				eMagazineOperation := E_MAGAZINE_OPERATION.TAKE;
				Diag.eState := E_CELL_STATE.MAGAZINE;
			ELSE
				Diag.eState := E_CELL_STATE.WAIT_MAGAZINE;
			END_IF;
		END_IF;

	E_CELL_STATE.SELECT_MACHINE:
		xCandidateFound := FALSE;
		xTimedCandidate := FALSE;
		uiSelectedMachine := 0;

		// Готовые станки выбираются по минимальному номеру.
		FOR uiLoop := 1 TO 3 DO
			IF NOT xCandidateFound
			AND astMachineStatus[uiLoop].xEnabled
			AND astMachineStatus[uiLoop].xCanAcceptService
			AND astMachineStatus[uiLoop].xServiceRequired
			AND NOT astMachineStatus[uiLoop].xError THEN
				uiSelectedMachine := uiLoop;
				xCandidateFound := TRUE;
			END_IF;
		END_FOR;

		IF xCandidateFound THEN
			Diag.eState := E_CELL_STATE.MOVE_TO_MACHINE;
		ELSE
			// Среди обрабатывающих станков выбирается минимальное оставшееся время.
			FOR uiLoop := 1 TO 3 DO
				IF astMachineStatus[uiLoop].xEnabled
				AND astMachineStatus[uiLoop].xProcessing
				AND astMachineStatus[uiLoop].xCycleTimeValid
				AND NOT astMachineStatus[uiLoop].xError THEN
					IF NOT xTimedCandidate
					OR (astMachineStatus[uiLoop].tRemaining < tMinimumRemaining) THEN
						uiSelectedMachine := uiLoop;
						tMinimumRemaining := astMachineStatus[uiLoop].tRemaining;
						xTimedCandidate := TRUE;
					END_IF;
				END_IF;
			END_FOR;

			// Без оценки времени ожидаем первый обрабатывающий станок.
			IF NOT xTimedCandidate THEN
				FOR uiLoop := 1 TO 3 DO
					IF (uiSelectedMachine = 0)
					AND astMachineStatus[uiLoop].xEnabled
					AND astMachineStatus[uiLoop].xProcessing
					AND NOT astMachineStatus[uiLoop].xError THEN
						uiSelectedMachine := uiLoop;
					END_IF;
				END_FOR;
			END_IF;

			IF uiSelectedMachine > 0 THEN
				Diag.eState := E_CELL_STATE.MOVE_TO_MACHINE;
			END_IF;
		END_IF;

	E_CELL_STATE.MOVE_TO_MACHINE:
		IF xStopRequested
		AND NOT stRobotStatus.xBusy THEN
			xRunning := FALSE;
			Diag.eState := E_CELL_STATE.IDLE;
		ELSIF (uiSelectedMachine < 1)
		OR (uiSelectedMachine > 3) THEN
			Diag.eState := E_CELL_STATE.SELECT_MACHINE;
		ELSIF NOT astMachineStatus[uiSelectedMachine].xEnabled
		OR astMachineStatus[uiSelectedMachine].xError THEN
			Diag.eState := E_CELL_STATE.SELECT_MACHINE;

		ELSIF stRobotStatus.eCurrentPoint = astMachineStatus[uiSelectedMachine].eAbovePoint THEN
			IF astMachineStatus[uiSelectedMachine].xCanAcceptService THEN
				Diag.eState := E_CELL_STATE.SERVICE_MACHINE;
			ELSE
				Diag.eState := E_CELL_STATE.WAIT_MACHINE;
			END_IF;

		ELSE
			Command.stRobot.xExecute := TRUE;
			Command.stRobot.eAction := E_ROBOT_ACTION.MOVE_TO_POINT;
			Command.stRobot.eSetPoint := astMachineStatus[uiSelectedMachine].eAbovePoint;

			IF stRobotStatus.xError THEN
				Error.dwErrorActive := Error.dwErrorActive OR ERR_ROBOT;
				Diag.eState := E_CELL_STATE.ERROR;
			ELSIF stRobotStatus.xDone THEN
				Diag.eState := E_CELL_STATE.RELEASE_ROBOT_COMMAND;
			END_IF;
		END_IF;

	E_CELL_STATE.RELEASE_ROBOT_COMMAND:
		IF stRobotStatus.xError THEN
			Error.dwErrorActive := Error.dwErrorActive OR ERR_ROBOT;
			Diag.eState := E_CELL_STATE.ERROR;
		ELSIF NOT stRobotStatus.xBusy
		AND NOT stRobotStatus.xDone THEN
			IF xStopRequested THEN
				xRunning := FALSE;
				Diag.eState := E_CELL_STATE.IDLE;
			ELSIF astMachineStatus[uiSelectedMachine].xCanAcceptService THEN
				Diag.eState := E_CELL_STATE.SERVICE_MACHINE;
			ELSE
				Diag.eState := E_CELL_STATE.WAIT_MACHINE;
			END_IF;
		END_IF;

	E_CELL_STATE.WAIT_MACHINE:
		IF NOT astMachineStatus[uiSelectedMachine].xEnabled
		OR astMachineStatus[uiSelectedMachine].xError THEN
			Diag.eState := E_CELL_STATE.SELECT_MACHINE;
		ELSIF astMachineStatus[uiSelectedMachine].xCanAcceptService THEN
			IF stRobotStatus.eCurrentPoint = astMachineStatus[uiSelectedMachine].eAbovePoint THEN
				Diag.eState := E_CELL_STATE.SERVICE_MACHINE;
			ELSE
				Diag.eState := E_CELL_STATE.MOVE_TO_MACHINE;
			END_IF;
		END_IF;

	E_CELL_STATE.SERVICE_MACHINE:
		IF xStopRequested
		AND NOT astMachineStatus[uiSelectedMachine].xBusy THEN
			xRunning := FALSE;
			Diag.eState := E_CELL_STATE.IDLE;
		ELSE
			Command.axMachineExecute[uiSelectedMachine] := TRUE;
		END_IF;

		IF Diag.eState = E_CELL_STATE.SERVICE_MACHINE THEN
			IF astMachineStatus[uiSelectedMachine].xError THEN
				Error.dwErrorActive := Error.dwErrorActive OR ERR_MACHINE;
				Diag.eState := E_CELL_STATE.ERROR;
			ELSIF stRobotStatus.xError THEN
				Error.dwErrorActive := Error.dwErrorActive OR ERR_ROBOT;
				Diag.eState := E_CELL_STATE.ERROR;
			ELSIF astMachineStatus[uiSelectedMachine].xRobotReleased THEN
				IF xStopRequested THEN
					xRunning := FALSE;
					Diag.eState := E_CELL_STATE.IDLE;
				ELSE
					Diag.eState := E_CELL_STATE.ROUTE_PAYLOAD;
				END_IF;
			END_IF;
		END_IF;

	E_CELL_STATE.MAGAZINE:
		IF xStopRequested
		AND NOT stMagazineStatus.xBusy THEN
			xRunning := FALSE;
			Diag.eState := E_CELL_STATE.IDLE;
		ELSE
			Command.stMagazine.xExecute := TRUE;
		END_IF;

		IF Diag.eState = E_CELL_STATE.MAGAZINE THEN
			IF stMagazineStatus.xError THEN
				Error.dwErrorActive := Error.dwErrorActive OR ERR_MAGAZINE;
				Diag.eState := E_CELL_STATE.ERROR;
			ELSIF stRobotStatus.xError THEN
				Error.dwErrorActive := Error.dwErrorActive OR ERR_ROBOT;
				Diag.eState := E_CELL_STATE.ERROR;
			ELSIF stMagazineStatus.xDone THEN
				Diag.eState := E_CELL_STATE.RELEASE_MAGAZINE;
			END_IF;
		END_IF;

	E_CELL_STATE.RELEASE_MAGAZINE:
		IF stMagazineStatus.xError THEN
			Error.dwErrorActive := Error.dwErrorActive OR ERR_MAGAZINE;
			Diag.eState := E_CELL_STATE.ERROR;
		ELSIF NOT stMagazineStatus.xBusy
		AND NOT stMagazineStatus.xDone THEN
			eMagazineOperation := E_MAGAZINE_OPERATION.NONE;
			IF xStopRequested THEN
				xRunning := FALSE;
				Diag.eState := E_CELL_STATE.IDLE;
			ELSE
				Diag.eState := E_CELL_STATE.ROUTE_PAYLOAD;
			END_IF;
		END_IF;

	E_CELL_STATE.WAIT_MAGAZINE:
		IF stMagazineStatus.xError THEN
			Error.dwErrorActive := Error.dwErrorActive OR ERR_MAGAZINE;
			Diag.eState := E_CELL_STATE.ERROR;
		ELSIF stMagazineStatus.xEnabled
		AND stRobotStatus.xDetailAvailable
		AND (stMagazineStatus.xCanChange OR stMagazineStatus.xCanPut) THEN
			Diag.eState := E_CELL_STATE.ROUTE_PAYLOAD;
		ELSIF stMagazineStatus.xEnabled
		AND NOT stRobotStatus.xBlankAvailable
		AND NOT stRobotStatus.xDetailAvailable
		AND stMagazineStatus.xCanTake THEN
			Diag.eState := E_CELL_STATE.ROUTE_PAYLOAD;
		END_IF;

	E_CELL_STATE.ERROR:
		xRunning := FALSE;
		IF stRobotStatus.xBusy THEN
			Command.stRobot.xStop := TRUE;
		END_IF;
		IF stMagazineStatus.xBusy THEN
			Command.stMagazine.xStop := TRUE;
		END_IF;

		IF xReset
		AND NOT xGlobalError
		AND NOT stRobotStatus.xError
		AND NOT stMagazineStatus.xError THEN
			Error.dwErrorLast := Error.dwErrorActive;
			Error.dwErrorActive := DWORD#0;
			uiSelectedMachine := 0;
			eMagazineOperation := E_MAGAZINE_OPERATION.NONE;
			Diag.eState := E_CELL_STATE.IDLE;
		END_IF;
END_CASE;

Status.xRunning := xRunning;
Status.xBusy := xRunning
	AND (Diag.eState <> E_CELL_STATE.IDLE)
	AND (Diag.eState <> E_CELL_STATE.ERROR);
Status.xWaitingMachine := Diag.eState = E_CELL_STATE.SELECT_MACHINE
	OR Diag.eState = E_CELL_STATE.WAIT_MACHINE;
Status.xWaitingMagazine := Diag.eState = E_CELL_STATE.WAIT_MAGAZINE;
Status.xError := Diag.eState = E_CELL_STATE.ERROR;
Status.xReadyToStart := xReadyToStart;
Status.xDrivesReady := xDrivesReady;
Status.xRobotReady := xRobotReady;
Status.xMagazineReady := xMagazineReady;
Status.uiReadyMachines := uiReadyMachines;
Status.uiSelectedMachine := uiSelectedMachine;
Status.eMagazineOperation := eMagazineOperation;
Error.dwAlarmActive := Error.dwErrorActive AND ERR_BOTH_GRIPPERS;

IF Error.dwErrorActive <> DWORD#0 THEN
	Error.dwErrorLast := Error.dwErrorActive;
END_IF;

Error.stErrorActive := UpdateErrorView(dwError := Error.dwErrorActive);
Error.stErrorLast := UpdateErrorView(dwError := Error.dwErrorLast);
